REGION Network 13: Реле безопастности К21 группа 221,222,224,225,231-235,311,312,313-317
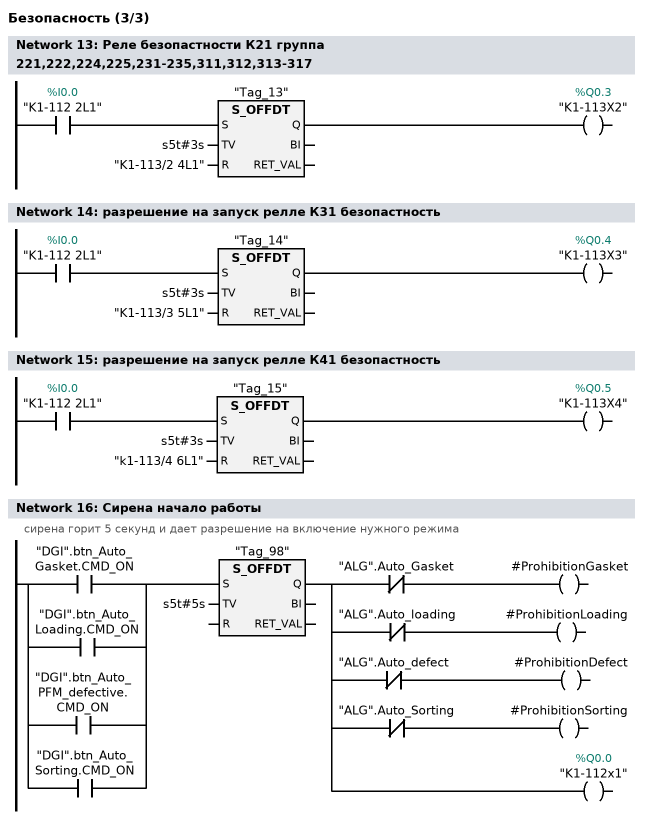
   RUNG wire#powerrail
      Contact( "K1-112 2L1" )
      S_OFFDT(T_NO := "Tag_13", TV := s5t#3s, R := "K1-113/2 4L1", BI =>, RET_VAL =>)
      Coil( "K1-113X2" )
   END_RUNG
   // the same network as SCL:
   #_s5time1 := S_OFFDT(T_NO := "Tag_13", S := "K1-112 2L1", TV := s5t#3s, R := "K1-113/2 4L1", Q => #_w1);
   "K1-113X2" := #_w1;
END_REGION

REGION Network 14: разрешение на запуск релле К31 безопастность
   RUNG wire#powerrail
      Contact( "K1-112 2L1" )
      S_OFFDT(T_NO := "Tag_14", TV := s5t#3s, R := "K1-113/3 5L1", BI =>, RET_VAL =>)
      Coil( "K1-113X3" )
   END_RUNG
   // the same network as SCL:
   #_s5time1 := S_OFFDT(T_NO := "Tag_14", S := "K1-112 2L1", TV := s5t#3s, R := "K1-113/3 5L1", Q => #_w1);
   "K1-113X3" := #_w1;
END_REGION

REGION Network 15: разрешение на запуск релле К41 безопастность
   RUNG wire#powerrail
      Contact( "K1-112 2L1" )
      S_OFFDT(T_NO := "Tag_15", TV := s5t#3s, R := "k1-113/4 6L1", BI =>, RET_VAL =>)
      Coil( "K1-113X4" )
   END_RUNG
   // the same network as SCL:
   #_s5time1 := S_OFFDT(T_NO := "Tag_15", S := "K1-112 2L1", TV := s5t#3s, R := "k1-113/4 6L1", Q => #_w1);
   "K1-113X4" := #_w1;
END_REGION

REGION Network 16: Сирена начало работы
   // сирена горит 5 секунд и дает разрешение на включение нужного режима
   RUNG wire#powerrail
      Contact( "DGI".btn_Auto_Gasket.CMD_ON )
      wire#w1
      S_OFFDT(T_NO := "Tag_98", TV := s5t#5s, R :=, BI =>, RET_VAL =>)
      wire#w2
      I_Contact( "ALG".Auto_Gasket )
      Coil( #ProhibitionGasket )
   END_RUNG
   RUNG wire#powerrail
      Contact( "DGI".btn_Auto_Loading.CMD_ON )
   END_RUNG wire#w1
   RUNG wire#powerrail
      Contact( "DGI".btn_Auto_PFM_defective.CMD_ON )
   END_RUNG wire#w1
   RUNG wire#powerrail
      Contact( "DGI".btn_Auto_Sorting.CMD_ON )
   END_RUNG wire#w1
   RUNG wire#w2
      I_Contact( "ALG".Auto_loading )
      Coil( #ProhibitionLoading )
   END_RUNG
   RUNG wire#w2
      I_Contact( "ALG".Auto_defect )
      Coil( #ProhibitionDefect )
   END_RUNG
   RUNG wire#w2
      I_Contact( "ALG".Auto_Sorting )
      Coil( #ProhibitionSorting )
   END_RUNG
   RUNG wire#w2
      Coil( "K1-112x1" )
   END_RUNG
   // the same network as SCL:
   #_s5time1 := S_OFFDT(T_NO := "Tag_98",
                        S := "DGI".btn_Auto_Gasket.CMD_ON OR "DGI".btn_Auto_Loading.CMD_ON OR "DGI".btn_Auto_PFM_defective.CMD_ON OR "DGI".btn_Auto_Sorting.CMD_ON,
                        TV := s5t#5s,
                        Q => #_w1);
   #ProhibitionGasket := #_w1 AND NOT "ALG".Auto_Gasket;
   #ProhibitionLoading := #_w1 AND NOT "ALG".Auto_loading;
   #ProhibitionDefect := #_w1 AND NOT "ALG".Auto_defect;
   #ProhibitionSorting := #_w1 AND NOT "ALG".Auto_Sorting;
   "K1-112x1" := #_w1;
END_REGION
END_FUNCTION_BLOCK

FUNCTION_BLOCK "FB_Link_Server"
{ S7_Optimized_Access := 'FALSE' }
VERSION : 0.1
   VAR 
      OperatorDetected : Bool;   // Можно начинать пересортировку оператор начал смену
      PackResortedReaded : Bool;   //     Пересортированный пакет прочитан
      FinishPackResorting : Bool;   //     Принудительно закончить пересортировку пакета
      Enable2Sxema : Bool;   // Собрать пакет 2мя схемами прокладок
      EnableRolling : Bool;   // Раскатать доски пакета на заданную длину
      SettingsWasApplyied : Bool;   // Были применены новые  настройки
      CheckPlankL : Bool;   // Проверять длину доски
      FinishDefectPack : Bool;   // Принудительно закончить сборку пакета  ПФМ брака
      DefectPacketPushed : Bool;   // пакет на ПФМ брака забрали
      PackDefectReaded : Bool;   // пакет на ПФМ брака прочитан сервером 
      PackParamChanged : Bool;   // Изменить параметры пакета
      PackReadyRidOff : Bool;   // пакет готов к выкатке
      GasketRidedOff : Bool;   // прокладку забрали с рамы
      PackToPack : Bool;   // режим из пакета в пакет
      AddGasketLayer : Bool;   // еще слой прокладки
      PackBrakParamChanged : Bool;   // корректировка параметров пакета брака
      QPlankLayers : Int;   // Количество слоев в пакете
      VPlanksInPack : Int;   //     Объём досок в пакете, м3
      QPlanksInLayer : Int;   //     Кол-во досок в слое досок пакета, шт
      QPlanksInLayerBrak : Int;   //     Кол-во досок в слое досок пакета брака, шт
      QPLankLayersBrak : Int;   //  Кол-во слоёв в пакете брака, шт
      Sxema : DInt;   //   Схема укладки прокладок
      SxemaNum : Int;   //     Номер схемы укладок прокладок
      PlankW : Int;   //     Ширина доски, мм
      PlankT : Int;   //     Толщина доски, мм
      Sxema2 : DInt;   // Cхема 2 укладки прокладок
      Sxema2Qlayers : Int;   //  Кол-во слоёв схемы 2 укладки прокладок
      PackL : Int;   // Длина пересобираемого пакета
      PartId : DInt;   // Ключ к пересобираемой партии (на случай перезапуска сервака)
      PlankL : Int;   // проверяемая длина доски
      ItemId : DInt;   // Ключ к номенклатуре пакета (на случай перезапуска сервака)
      SetNumLayer : Int;   // Корректируемое кол-во уложенных слоев досокб шт
      SetNumPlankInLayer : Int;   // Коррктируемое кол-во досок в слоеб шт
      GeneralSpeed : Int := 50;   // Общая скорость линии
      TotalPlanksInPack : Int;   // всего досок в пакете
      SetNumPlanksInLayerBrak : Int;   // коррекция счета досок в слое брака
      CheckL : Int;   // проверяемая длина доски
      GasketBrakPut : Bool;   // положили бруски на пакет брака
      GasketLayersPeriod : Int;   // Периодичность брусков пакета брака
      LineInWork : Bool;   //     Линия в работе
      PackResorting : Bool;   //     Пакет пересортировывается
      PackResorted : Bool;   //     Пакет пересортировался
      PackBrakComplete : Bool;   //  Пакет брака собран
      RdyStartNewPack : Bool;   //     Есть готовность к пересборке нового пакета
      RdyStart : Bool;   //     Есть готовность к запуску линии
      DefectPacketResorted : Bool;   // Пакет на ПФМ брака пересортирован
      NumLayerActual : Int;   //     Текущее кол-во уложенных слоёв досок, шт
      NumPlanksInLayerActual : Int;   //     Текущее кол-во уложенных слоёв прокладок, шт
      QPlanksOk : Int;   //     Текущее кол-во уложенных досок, шт
      QPlanksNotOk : Int;   //     Текущее кол-во уложенных херовых досок, шт
      VPlanksOk : DInt;   //     Текущий объём уложенных досок, м3*1000
      QPlankBrak : Int;   // Кол-во досок в пакете брака
      VLayerOk : DInt;   // Объем собирающегося слоя, м3
      M_211 : "ServIM";   //      Загрузочный транспортёр
      M_212 : "ServIM";   //      Загрузочный лифт сортировки+тормоз
      M_213 : "ServIM";   //      Наклюнный транспортёр после лифта
      M_214 : "ServIM";   //      Приёмный транспортёр прокладок
      M_221 : "ServIM";   //      Горка основная
      M_222 : "ServIM";   //      Транспортёр цепной после элеватора
      M_223 : "ServIM";   //      Резерв
      M_224 : "ServIM";   //      Упоры поштучника
      M_225 : "ServIM";   //      Транспортёр бобышек
      M_231 : "ServIM";   //      Ролики торцовочные
      M_232 : "ServIM";   //      Лифт ПФМ
      M_233 : "ServIM";   //      Вилы ПФМ
      ForkRotator : "ServIM";   //  Поворот вилы основной ПФМ
      M_234 : "ServIM";   //      Тр-тёр прокладок перед крючками ПФМ
      M_235 : "ServIM";   //      Подвижной борт
      M_311 : "ServIM";   //      Ленточный тр-тёр удаления прокладок
      M_312 : "ServIM";   //      Горка прокладок 1
      M_313 : "ServIM";   //      Тр-тёр прокладок после горки прокладок 1
      M_314 : "ServIM";   //      Горка прокладок 2
      M_315 : "ServIM";   //      Горка прокладок 3
      M_316 : "ServIM";   //      Тр-тёр загрузки прокладок в горку 2
      M_317 : "ServIM";   //      Основной транспортёр прокладок
      GasketSupplier : "ServIM";   // Выдача прокладки на карусель
      M_321 : "ServIM";   //      Выкатной транспортёр ПФМ 1
      M_322 : "ServIM";   //      Выкатной транспортёр ПФМ 2
      M_323 : "ServIM";
      M_324 : "ServIM";   //      Выкатной транспортёр ПФМ 3 (выгрузка пакета)
      M_325 : "ServIM";   //  Транспортер приема доски с Горки перед поштучкой
      M_330 : "ServIM";   //  Ленточный транспортер брака
      M_331 : "ServIM";   //      Ленточный транспортёр брака
      M_332 : "ServIM";   //      Сбрасыватель с рольганга брака
      M_333 : "ServIM";   //      Рольганг брака
      M_334 : "ServIM";   //      Тр-тёр сбора слоя ПФМ брака
      M_335 : "ServIM";   //      Вилы ПФМ брака
      M_336 : "ServIM";   //      Лифт ПФМ брака
      Alarm_List { S7_SetPoint := 'True'} : Array[0..255] of Bool;
   END_VAR


BEGIN
	    //Сбросим задание на подвижный борт, после того как в FB_Link_Server он был взведен по новому заданию
	    "ALG".ModeChang := FALSE;
	    "ALG".ForceFinishMainPFM := FALSE;
	    "ALG".ForceFinishPFMDefect := FALSE;
	    "ALG".DefectivePacketIsPushed := FALSE;
	    "ALG".EmptyLodems := FALSE;
	    "ALG".AddGasketLayer := FALSE;
	    "ALG".ConfirmGasketsBrak := FALSE;
	    
	    //Пришел бит с сервера "Начать новый пакет" (вместе с прочими исходными данными)
	 //   IF #OperatorDetected THEN
	 //       #QPlanksNotOk := 0;
	 //       #QPlanksOk := 0;
	        
	        // В конце бит с сервера "Начать новый пакет" обнулим
	 //       #OperatorDetected := FALSE;
	 //   END_IF;
	    
	    //Ежели были применены новые настройки
	    IF #SettingsWasApplyied THEN
	        
	      // для подвижного борта
	        "ALG".ModeChang := true;
	        
	        // для определения задержки
	        "ALG".PermMovM323 := "SolveLinearDelay"(LinearParam:=#PlankW, Koef:=2.5, Offset:=10);
	        "ALG".SqueezeRamp := "SolveLinearDelay"(LinearParam := 60 - #PlankT,
	                                                Koef := 10.0,
	                                                Offset := 100);
	        
	        "ALG".SqueezeUporPFM := "SolveLinearDelay"(LinearParam := #PlankT,
	                                                   Koef := 3.75,
	                                                   Offset := 10);
	        
	        #PackResorted := FALSE;
	        
	        #RdyStartNewPack := False;
	        
	        #RdyStart := FALSE;
	        #SettingsWasApplyied := FALSE;
	        
	       
	    END_IF;
	    
	    
	    
	    //Пришел бит с сервера или кнопки "Принудительно завершить пересортировку пакета"
	    IF #FinishPackResorting THEN
	        
	        //...//
	        "ALG".ForceFinishMainPFM := TRUE;
	        
	        // В конце его обнулим
	        #FinishPackResorting := FALSE;
	    END_IF;
	    
	    //Пришел бит с сервера "Принудительно завершить пересортировку пакета брака"
	    IF #FinishDefectPack THEN
	        
	        //...//
	        "ALG".ForceFinishPFMDefect := TRUE;
	        
	        
	        // В конце его обнулим
	        #FinishDefectPack := FALSE;
	    END_IF;
	    
	    IF (#DefectPacketPushed) THEN
	        "ALG".DefectivePacketIsPushed := TRUE;
	        
	        #DefectPacketPushed := FALSE;
	    END_IF;
	    
	    // Пришел битяра, что пакет брака прочитан и записан в ДБ
	    IF (#PackDefectReaded) THEN
	        
	        #DefectPacketResorted := FALSE;
	        #QPlanksNotOk := 0;
	        
	        #PackDefectReaded := False;
	    END_IF;
	    
	    // Пришел бит на изменение кол-ва досок в слое, кол-во слоев в пакете
	    IF (#PackParamChanged) THEN
	        // если на раме прокладок сейчас ничего нет, то просто меняем внутренний счетчик
	        IF ( "Сортировка_DB".LayersCounter <> #SetNumLayer) THEN
	            IF ("FB_Ramp_DB".s_busy) THEN
	                "FB_Ramp_DB".layer_holded := #SetNumLayer + 1;
	            ELSE
	                "FB_Ramp_DB".layer_holded := #SetNumLayer;
	            END_IF;
	        END_IF;
	        
	        "Сортировка_DB".LayersCounter := #SetNumLayer;
	        "Сортировка_DB".BoardInLayerCounter := #SetNumPlankInLayer;
	        
	        
	        
	        #PackParamChanged := False;
	    END_IF;
	    
	    
	    // На пакет наклеили этикетку
	    IF (#PackReadyRidOff) THEN
	        // Переменная для работы логики фиксируется
	        "ALG".PacketReadyRollOut := "S16.1" AND "B18.0" AND "Сортировка_DB".LiftPushingPacket;
	        // сразу обнуляемся
	        #PackReadyRidOff := FALSE;
	    END_IF;
	    
	    //бит прокладочник очищен
	    IF (#GasketRidedOff) THEN
	        "ALG".EmptyLodems := TRUE;
	        
	        #GasketRidedOff := FALSE;
	    END_IF;
	    
	    // бит добавить еще слой прокладок
	    // 
	    IF (#AddGasketLayer) THEN
	        "ALG".AddGasketLayer := TRUE;
	        
	        #AddGasketLayer := FALSE;
	    END_IF;
	    
	    IF (#GasketBrakPut) THEN
	        "ALG".ConfirmGasketsBrak := "B22.6";
	        
	        #GasketBrakPut := FALSE;
	    END_IF;
	   
	    //
	    IF (#PackBrakParamChanged) THEN
	        "ПФМ Брака_DB".BoardsInLayCounter := #SetNumPlanksInLayerBrak;
	        
	        #PackBrakParamChanged := FALSE;
	    END_IF;
	    
	    //Пришел бит с сервера "Сервер прочитал что пакет пересобран" или бит "Принудительно завершить пересортировку пакета"
	    IF #PackResortedReaded THEN
	        
	        //...// 
	        
	        //Обнулим задание на пересборку пакета и актуальные значения
	(*        #NumGasketActual := 0;
	        #NumLayerActual := 0;
	        #PlankT := 0;
	        #PlankW := 0;
	        #Sxema := 0;
	        #QPlanksInLayerBrak := 0;
	        #QPlankLayers := 0;
	        #QPlanksInLayer := 0;
	        #QPlanksNotOk := 0;
	        #QPlanksOk := 0;
	        #SxemaNum := 0;
	        #VPlanksOk := 0;
	        #Sxema2 := 0;
	        #Sxema2Qlayers := 0;
	        #PackL := 0; *)
	        //#PackId := 0;
	        //
	        #QPlanksOk := 0;
	        "ALG".Volume := 0;
	        #VPlanksOk := 0;
	        
	        #PackResorted := FALSE;
	        
	        // В конце его обнулим
	        #PackResortedReaded := FALSE;
	    END_IF;
	    //==============================================================================================
	    //M211 Загрузочный транспортер пакета
	    
	    (* IF #M_211.BtnAU THEN
	        #M_211.BtnAU := FALSE;
	    END_IF;
	    IF #M_211.BtnDU THEN
	        #M_211.BtnDU := FALSE;
	    END_IF;
	    IF #M_211.BtnFwd THEN
	        #M_211.BtnFwd := FALSE;
	    END_IF;
	    IF #M_211.BtnBwd THEN
	        #M_211.BtnBwd := FALSE;
	    END_IF;
	    IF #M_211.BtnCmdStop THEN
	        #M_211.BtnCmdStop := FALSE;
	    END_IF;     
	    IF #M_211.BtnDU THEN
	        "IM".M_211_Load_Transp.btnDU := TRUE;
	        #M_211.BtnDU := FALSE;
	        
	    END_IF;*)
	    
	    
	    REGION Список аварий заполнение
	        // Motor faults
	        // 
	        #Alarm_List[0] := "IM".M_211_Load_Transp.notON;
	        #Alarm_List[1] := "IM".M_211_Load_Transp.notOFF;
	        #Alarm_List[2] := "IM".M_311_Strip_Remov.notON;
	        #Alarm_List[3] := "IM".M_311_Strip_Remov.notOFF;
	        #Alarm_List[4] := "IM".M_212_Sort_Elevator.notOn;
	        #Alarm_List[5] := "IM".M_212_Sort_Elevator.notCMD;
	        #Alarm_List[6] := "IM".M_212_Sort_Elevator.notOff;
	        #Alarm_List[7] := "IM".M_212_Sort_Elevator.wrong_state;
	        #Alarm_List[8] := "IM".M_212_Sort_Elevator.wrong_CMD;
	        #Alarm_List[9] := "IM".M_213_ConvElevator.notON;
	        #Alarm_List[10] := "IM".M_213_ConvElevator.notOFF;
	        #Alarm_List[11] := "IM".M_222_Main_Sort_Slide.notON;
	        #Alarm_List[12] := "IM".M_222_Main_Sort_Slide.notOFF;
	        #Alarm_List[13] := "IM".M_325_Tr_Hill.notON;
	        #Alarm_List[14] := "IM".M_325_Tr_Hill.notOFF;
	        #Alarm_List[15] := "IM".M_223_Evaluation_area.notON;
	        #Alarm_List[16] := "IM".M_223_Evaluation_area.notOFF;
	        #Alarm_List[17] := "IM".M_224_Individ_dispensing.notOn;
	        #Alarm_List[18] := "IM".M_224_Individ_dispensing.notCMD;
	        #Alarm_List[19] := "IM".M_224_Individ_dispensing.notOff;
	        #Alarm_List[20] := "IM".M_224_Individ_dispensing.wrong_state;
	        #Alarm_List[21] := "IM".M_224_Individ_dispensing.wrong_CMD;
	        #Alarm_List[22] := "IM".M_225_Conveyor_with_lugs.notON;
	        #Alarm_List[23] := "IM".M_225_Conveyor_with_lugs.notOFF;
	        #Alarm_List[24] := "IM".M_235_Movable_board.notOn;
	        #Alarm_List[25] := "IM".M_235_Movable_board.notCMD;
	        #Alarm_List[26] := "IM".M_235_Movable_board.notOff;
	        #Alarm_List[27] := "IM".M_235_Movable_board.wrong_state;
	        #Alarm_List[28] := "IM".M_235_Movable_board.wrong_CMD;
	        #Alarm_List[29] := "IM".M_231_Roller_conveyor.notON;
	        #Alarm_List[30] := "IM".M_231_Roller_conveyor.notOFF;
	        #Alarm_List[31] := "IM".M_323_Small_Chain.notON;
	        #Alarm_List[32] := "IM".M_323_Small_Chain.notOFF;
	        #Alarm_List[33] := "IM".M_214_Gasket_receiver.notON;
	        #Alarm_List[34] := "IM".M_214_Gasket_receiver.notOFF;
	        #Alarm_List[35] := "IM".M_312_First_slide.notON;
	        #Alarm_List[36] := "IM".M_312_First_slide.notOFF;
	        #Alarm_List[37] := "IM".M_313_AF_slide_conv.notON;
	        #Alarm_List[38] := "IM".M_313_AF_slide_conv.notOFF;
	        #Alarm_List[39] := "IM".M_316_Padloader_IN2.notON;
	        #Alarm_List[40] := "IM".M_316_Padloader_IN2.notOFF;
	        #Alarm_List[41] := "IM".M_314_Second_slide.notON;
	        #Alarm_List[42] := "IM".M_314_Second_slide.notOFF;
	        #Alarm_List[43] := "IM".M_315_Third_slide.notON;
	        #Alarm_List[44] := "IM".M_315_Third_slide.notOFF;
	        #Alarm_List[45] := "IM".M_234_Carousel_loader.notON;
	        #Alarm_List[46] := "IM".M_234_Carousel_loader.notOFF;
	        #Alarm_List[47] := "IM".M_330_Scrap_Conv.notON;
	        #Alarm_List[48] := "IM".M_330_Scrap_Conv.notOFF;
	        #Alarm_List[49] := "IM".M_331_Scrap_conveyor.notON;
	        #Alarm_List[50] := "IM".M_331_Scrap_conveyor.notOFF;
	        #Alarm_List[51] := "IM".M_332_Dump_lug_conv.notON;
	        #Alarm_List[52] := "IM".M_332_Dump_lug_conv.notOFF;
	        #Alarm_List[53] := "IM".M_333_Defective_roller.notON;
	        #Alarm_List[54] := "IM".M_333_Defective_roller.notOFF;
	        #Alarm_List[55] := "IM".M_334_Layer_set_conv.notON;
	        #Alarm_List[56] := "IM".M_334_Layer_set_conv.notOFF;
	        #Alarm_List[57] := "IM".M_335_Lay_fork_scrap.notON;
	        #Alarm_List[58] := "IM".M_335_Lay_fork_scrap.notOFF;
	        #Alarm_List[59] := "IM".M_335_Lay_fork_scrap.notCMD;
	        #Alarm_List[60] := "IM".M_335_Lay_fork_scrap.notFeedBack;
	        #Alarm_List[61] := "IM".M_335_Lay_fork_scrap.wrong_state;
	        #Alarm_List[62] := "IM".M_336_PFM_elevator.notOn;
	        #Alarm_List[63] := "IM".M_336_PFM_elevator.notCMD;
	        #Alarm_List[64] := "IM".M_336_PFM_elevator.notOff;
	        #Alarm_List[65] := "IM".M_336_PFM_elevator.wrong_state;
	        #Alarm_List[66] := "IM".M_336_PFM_elevator.wrong_CMD;
	        #Alarm_List[67] := "IM_Rout".M_321_Rollgang_Lift_PFM.notON;
	        #Alarm_List[68] := "IM_Rout".M_321_Rollgang_Lift_PFM.notOFF;
	        #Alarm_List[69] := "IM_Rout".M_322_Conveyor_2.notON;
	        #Alarm_List[70] := "IM_Rout".M_322_Conveyor_2.notOFF;
	        #Alarm_List[71] := "IM_Rout".M_324_Rout_Conveyor.notON;
	        #Alarm_List[72] := "IM_Rout".M_324_Rout_Conveyor.notOFF;
	        #Alarm_List[73] := "IM_PFM".M_233_Fork_PFM.notON;
	        #Alarm_List[74] := "IM_PFM".M_233_Fork_PFM.notOFF;
	        #Alarm_List[75] := "IM_PFM".M_233_Fork_PFM.notCMD;
	        #Alarm_List[76] := "IM_PFM".M_233_Fork_PFM.notFeedBack;
	        #Alarm_List[77] := "IM_PFM".M_232_Elevator_PFM.notOn;
	        #Alarm_List[78] := "IM_PFM".M_232_Elevator_PFM.notCMD;
	        #Alarm_List[79] := "IM_PFM".M_232_Elevator_PFM.notOff;
	        #Alarm_List[80] := "IM_PFM".M_232_Elevator_PFM.wrong_state;
	        #Alarm_List[81] := "IM_PFM".M_232_Elevator_PFM.wrong_CMD;
	        #Alarm_List[82] := "IM_PFM".M_317_Gasket_Carousel.notON;
	        #Alarm_List[83] := "IM_PFM".M_317_Gasket_Carousel.notOFF;
	        #Alarm_List[84] := "HS".Gasket_Ramp.notUp;
	        #Alarm_List[85] := "HS".Gasket_Ramp.notMid;
	        #Alarm_List[86] := "HS".Gasket_Ramp.notDn;
	        #Alarm_List[87] := "HS".Gasket_Ramp.wrong_state;
	        #Alarm_List[88] := "HS".Gasket_Ramp.wrong_CMD;
	        #Alarm_List[89] := "HS".Gasket_Lodems.notON;
	        #Alarm_List[90] := "HS".Gasket_Lodems.notOFF;
	        #Alarm_List[91] := "HS".Gasket_Lodems.notCMD;
	        #Alarm_List[92] := "HS".Gasket_Lodems.notFeedBack;
	        #Alarm_List[93] := "HS".Gasket_Lodems.wrong_state;
	        #Alarm_List[94] := "HS".Forks_Pitcher.notON;
	        #Alarm_List[95] := "HS".Forks_Pitcher.notOFF;
	        #Alarm_List[96] := "HS".Forks_Pitcher.notCMD;
	        #Alarm_List[97] := "HS".Forks_Pitcher.notFeedBack;
	        #Alarm_List[98] := "HS".Forks_Pitcher.wrong_state;
	        #Alarm_List[99] := "HS".Upor_Defective.notON;
	        #Alarm_List[100] := "HS".Upor_Defective.notOFF;
	        #Alarm_List[101] := "HS".Upor_Defective.notCMD;
	        #Alarm_List[102] := "HS".Upor_Defective.notFeedBack;
	        #Alarm_List[103] := "HS".Upor_Defective.wrong_state;
	        #Alarm_List[104] := "HS".M_221_Large_HydroStationDrive.notOn;
	        #Alarm_List[105] := "HS".M_221_Large_HydroStationDrive.notOff;
	        #Alarm_List[106] := "HS".M_221_Large_HydroStationDrive.wrongValveState;
	        #Alarm_List[107] := "HS".M_337_Small_HydroStationDrive.notOn;
	        #Alarm_List[108] := "HS".M_337_Small_HydroStationDrive.notOff;
	        #Alarm_List[109] := "HS".M_337_Small_HydroStationDrive.wrongValveState;
	        
	        
	        // Logic faults
	        // 
	        #Alarm_List[110] := "QueueController_DB".AlarmWrongLength;
	        #Alarm_List[111] := "FB_Gasket_Carousel_DB".s_paused; // "FB_SetGaskets_DB".Paused;
	        #Alarm_List[112] := "FB_Gasket_Carousel_DB".ALM_NoGasketToUP;  // "FB_SetGaskets_DB".ALM_NoGasketToUP;
	        #Alarm_List[113] := "EvaluationZoneThrowOFF_DB".AlarmBoardNotExitFromZone;
	        #Alarm_List[114] := "Сортировка_DB".AlarmLowerElevator;
	        #Alarm_List[115] := "UporPFM_DB".AlarmGidra; // уберите доску после упоров ПФМ
	        #Alarm_List[116] := "UporPFM_DB".AlarmWarpingBoard; // уберите доску после упоров ПФМ
	        
	        // Sxema Faults
	        // 
	        
	        #Alarm_List[117] := "QueueController_DB".AlarmNotValidHole AND NOT "QueueController_DB".Hint_3;  // Ожидался пробел между слоями, уберите доску под линейкой, следующая доска должна быть на низкой цепи
	        #Alarm_List[118] := "QueueController_DB".AlarmNotValidHole AND "QueueController_DB".Hint_3;
	        
	        #Alarm_List[119] := "QueueController_DB".AlarmNotAwaitableBoard AND "QueueController_DB".Hint_3 AND NOT "QueueController_DB".Hint_2; // не та доска под линейкой, переложите на след бобышку, следующая цепь высокая (Далее ожидается доска на высокой цепи)
	        #Alarm_List[120] := "QueueController_DB".AlarmNotAwaitableBoard AND "QueueController_DB".Hint_3  AND "QueueController_DB".Hint_2; // под линейкой ожидалась доска на высокой цепи, уберите доску
	        #Alarm_List[121] := "QueueController_DB".AlarmNotAwaitableBoard AND NOT "QueueController_DB".Hint_3  AND "QueueController_DB".Hint_2; // под линейкой ожидалась доска на низкой цепи, уберите доску
	        
	        #Alarm_List[122] := "QueueController_DB".AlarmNotAwaitableBoard AND NOT "QueueController_DB".Hint_3 AND NOT "QueueController_DB".Hint_2; // не та доска под линейкой, переложите на след бобышку, следующая цепь низкая Далее ожидается доска на низкой цепи)
	        
	        // SensLineAlarm
	        // 
	        #Alarm_List[123] := "SensorLine_Clogging_DB".AlarmSensor_dirty[0]; //загрязнен датчик 1,8 м
	        #Alarm_List[124] := "SensorLine_Clogging_DB".AlarmSensor_dirty[1];
	        #Alarm_List[125] := "SensorLine_Clogging_DB".AlarmSensor_dirty[2];
	        #Alarm_List[126] := "SensorLine_Clogging_DB".AlarmSensor_dirty[3];
	        #Alarm_List[127] := "SensorLine_Clogging_DB".AlarmSensor_dirty[4];
	        #Alarm_List[128] := "SensorLine_Clogging_DB".AlarmSensor_dirty[5];
	        #Alarm_List[129] := "SensorLine_Clogging_DB".AlarmSensor_dirty[6];
	        #Alarm_List[130] := "SensorLine_Clogging_DB".AlarmSensor_dirty[7];
	        #Alarm_List[131] := "SensorLine_Clogging_DB".AlarmSensor_dirty[8];
	        #Alarm_List[132] := "SensorLine_Clogging_DB".AlarmSensor_dirty[9];
	        #Alarm_List[133] := "SensorLine_Clogging_DB".AlarmSensor_dirty[10];
	        #Alarm_List[134] := "SensorLine_Clogging_DB".AlarmSensor_dirty[11];
	        #Alarm_List[135] := "SensorLine_Clogging_DB".AlarmSensor_dirty[12];
	        #Alarm_List[136] := "SensorLine_Clogging_DB".AlarmSensor_dirty[13];
	        #Alarm_List[137] := "SensorLine_Clogging_DB".AlarmSensor_dirty[14]; // загрязнен датчик 6.0 м
	        
	        //Sensor alarms
	        //
	        
	        
	        //MOOOre alarms
	        // 
	        #Alarm_List[138] := "IM_PFM".M_233_Fork_PFM.unkn_state; // вилы ПФМ в некорректном положении
	        #Alarm_List[139] := "EvaluationZoneThrowOFF_DB".FaultGhostBoard; // ошибка очереди на зоне оценки
	        #Alarm_List[140] := NOT "QueueController_DB".Calibrated; // линейка не откалибрована
	        #Alarm_List[141] := "Сортировка_DB".AlarmNotReadedPack; // ошибка чтения пакета ПФМ
	        #Alarm_List[142] := "ПФМ Брака_DB".AlarmNotReadedPack; // ошибка чтения пакета ПФМ брака
	        #Alarm_List[143] := "ПФМ Брака_DB".AlarmExtraBoardInLay; //ошибка лишняя доска на слой пфм брака
	        #Alarm_List[144] := "FB_Gasket_Carousel_DB".ALM_SensLastHook;  // "FB_SetGaskets_DB".ALM_LargeOffset; // ошибка переезда карусели
	        #Alarm_List[145] := "FB_Gasket_Carousel_DB".ALM_SensHook; // "FB_SetGaskets_DB".ALM_SensHook; // сбой датчика крюков на карусели
	        #Alarm_List[146] := "QueueController_DB".AlarmCount; // ошибка счета ПФМ
	        #Alarm_List[147] := "ПФМ Брака_DB".AlarmNoPacketPushed; //авария не забрали пакет с пфм брака
	        #Alarm_List[148] := "ПФМ Брака_DB".AwaitGasket; // ожидаем прокладку на пфм брака
	        
	        
	    END_REGION
	    
	
END_FUNCTION_BLOCK

FUNCTION "SolveLinearDelay" : Time
{ S7_Optimized_Access := 'FALSE' }
VERSION : 0.1
   VAR_INPUT 
      LinearParam : Int;   // линейный параметр
      Koef : Real;   // коэффициент k
      Offset : Int;   // коэффициент сдвига b
   END_VAR

   VAR_TEMP 
      Delay_in_ms : Real;
   END_VAR


BEGIN
	#Delay_in_ms := INT_TO_REAL(#LinearParam);
	
	#SolveLinearDelay := DINT_TO_TIME(TRUNC_DINT(#Koef * #Delay_in_ms) + #Offset);
END_FUNCTION

FUNCTION "GetGeneralSpeed" : Real
{ S7_Optimized_Access := 'FALSE' }
VERSION : 0.1
   VAR_INPUT 
      GS_from_Server : Int;
   END_VAR


BEGIN
	IF (#GS_from_Server < 10.0) THEN
	    #GetGeneralSpeed := 10.0;
	ELSE
	    #GetGeneralSpeed := INT_TO_REAL(#GS_from_Server);
	END_IF;
	
END_FUNCTION

FUNCTION_BLOCK "FB_Load_Zone"
{ S7_Optimized_Access := 'FALSE' }
VERSION : 0.1
   VAR 
      auto_mode_trigger : Bool;
      M213_mode : Bool;
      up_cmd_old : Bool;
      down_cmd_old : Bool;
      Lift_State : Int;
      Memento_Lift_State : Int;
      delayStart {InstructionName := 'TON'; LibVersion := '1.0'} : TON;
      wait_1 {InstructionName := 'TOF'; LibVersion := '1.0'} : TOF;
      wait_2 {InstructionName := 'TOF'; LibVersion := '1.0'} : TOF;
      wait_3 {InstructionName := 'TOF'; LibVersion := '1.0'} : TOF;
      wait_213 {InstructionName := 'TOF'; LibVersion := '1.0'} : TOF;
   END_VAR

   VAR_TEMP 
      Lift_UP : Bool;
      Lift_DOWN : Bool;
      Cancel_UP : Bool;
      Resume_UP : Bool;
      Sert : Word;
   END_VAR

   VAR CONSTANT 
      LIFT_WAITING : Int := 0;
      LIFT_START : Int := 1;
      LIFT_CYCLE : Int := 2;
      LIFT_RETURN : Int := 3;
      LIFT_STOP : Int := 4;
      LIFT_CANCEL : Int := 5;
      LIFT_UNKNOWN : Int := 10;
      DELAY_START : Time := T#5s;
   END_VAR


BEGIN
	REGION Ready and alarms LOADING ZONE
	    
	    "ALG".Ready_loading := "NaprUpr" AND "K1-113/1 3L1" AND "K1-112 2L1";
	  
	    "ALG".Alarm_loading :=
	    // Транспортер загрузки
	    "IM".M_211_Load_Transp.Alarm OR
	    "IM".M_211_Load_Transp.Fault OR
	    // Лифт Melektra
	    "IM".M_212_Sort_Elevator.Fault OR
	    // Наклонный транспортер
	    "IM".M_213_ConvElevator.Fault OR
	    "IM".M_213_ConvElevator.Alarm OR
	    // Транспортер прокладок
	    "IM".M_214_Gasket_receiver.Fault OR
	    "IM".M_214_Gasket_receiver.Alarm OR
	    // ??
	    "IM".M_311_Strip_Remov.Fault OR
	    // НЕТ СИГНАЛА ГОТОВОСТИ
	    NOT "ALG".Ready_loading
	    ;
	    
	END_REGION
	
	REGION Mode selector
	    
	    #auto_mode_trigger := (#auto_mode_trigger
	    OR
	    (
	    "DGI".btn_Auto_Loading.CMD_ON
	    ))
	    AND NOT
	    (
	    NOT "ALG".Ready_loading OR
	    "DGI".btn_Auto_Loading.CMD_OFF
	    );
	    
	    // State lamps
	    // 
	    "H76.3" := "H78.0" := #auto_mode_trigger;
	    
	    // Auto SIGNAL
	    "ALG".Auto_loading := #auto_mode_trigger AND NOT "Безопасность_DB".ProhibitionLoading;
	    
	END_REGION
	
	REGION M211
	    // Backwards
	    "IM".M_211_Load_Transp.btn_Back_ON := "E82.2";
	    
	    // Forward
	    "IM".M_211_Load_Transp.OnCom :=
	    
	    "S81.1"
	    OR
	    ("IM".M_211_Load_Transp.btn_Back_ON)
	    ;
	    
	    
	END_REGION
	
	REGION M212
	    // SIGNALS
	    // 
	    #Cancel_UP := "DGI".E82_5 AND NOT #down_cmd_old;
	    #Resume_UP := "DGI".S82_4 AND NOT #up_cmd_old;
	    
	    #up_cmd_old := "DGI".S82_4;
	    #down_cmd_old := "DGI".E82_5;
	    
	    // таймера
	    // 
	    #delayStart(IN := "koncevik2",
	                PT := #DELAY_START);
	    
	    #wait_1(IN := "nakloniy transporter",
	            PT := T#6s);
	    
	    #wait_2(IN := NOT "doska v priymke elevator",
	            PT := T#3s);
	    
	    #wait_3(IN := "sloi doski",
	            PT := T#6s);
	    
	    
	    // запуск лифта
	    CASE #Lift_State OF
	        // ожидание пакета
	        #LIFT_WAITING:
	            
	            // LOGIC
	            #Lift_UP := #Lift_DOWN := FALSE;
	            //"IM".M_212_Sort_Elevator.comUp := "IM".M_212_Sort_Elevator.comDown := FALSE;
	            
	            // Transitions
	            IF (#delayStart.Q) THEN
	                #Lift_State := #LIFT_START;
	                GOTO EndAutomata;
	            END_IF;
	            
	            IF (NOT "Lift Down") THEN
	                #Lift_State := #LIFT_CANCEL;
	            END_IF;
	            
	        #LIFT_START:
	            
	            // LOGIC
	            // 
	            #Lift_UP := TRUE;
	            #Lift_DOWN := FALSE;
	            //"IM".M_212_Sort_Elevator.comUp := #delayStart.Q;
	            //"IM".M_212_Sort_Elevator.comDown := False;
	            
	            // Transitions
	            IF ("sloi doski") THEN
	                #Lift_State := #LIFT_CYCLE;
	                GOTO EndAutomata;
	            END_IF;
	            
	            IF ("Lift Upp") THEN
	                #Lift_State := #LIFT_RETURN;
	            END_IF;
	            
	            IF (#Cancel_UP) THEN
	                #Memento_Lift_State := #Lift_State;
	                #Lift_State := #LIFT_STOP;
	            END_IF;
	            
	        #LIFT_CYCLE:
	            // LOGIC
	            // 
	            #Lift_DOWN := FALSE;
	            #Lift_UP := NOT (#wait_1.Q OR #wait_2.Q OR #wait_3.Q) OR "DGI".S82_4;
	            
	            // Transitions
	            IF ("Lift Upp") THEN
	                #Lift_State := #LIFT_RETURN;
	            END_IF;
	            
	            IF (#Cancel_UP) THEN
	                #Memento_Lift_State := #Lift_State;
	                #Lift_State := #LIFT_STOP;
	            END_IF;
	            
	        #LIFT_RETURN:
	            // LOGIC
	            #Lift_DOWN := TRUE;
	            #Lift_UP := FALSE;
	            
	            // Transitions
	            IF ("Lift Down") THEN
	                #Lift_State := #LIFT_WAITING;
	                GOTO EndAutomata;
	            END_IF;
	            
	        #LIFT_STOP:
	            // LOGIC;
	            // 
	            #Lift_DOWN := FALSE;
	            #Lift_UP := False;
	            
	            // Transitions
	            // 
	            IF (#Cancel_UP) THEN
	                #Lift_State := #LIFT_CANCEL;
	                GOTO EndAutomata;
	            END_IF;
	            
	            IF (#Resume_UP) THEN
	               
	                #Lift_State := #Memento_Lift_State;
	                
	            END_IF;
	            
	        #LIFT_CANCEL:
	            // LOGIC
	            #Lift_DOWN := TRUE;
	            #Lift_UP := FALSE;
	            
	            // Transitions
	            IF ("Lift Down") THEN
	                #Lift_State := #LIFT_WAITING;
	                GOTO EndAutomata;
	            END_IF;
	
	        ELSE  // Lift unknown state
	            ;
	    END_CASE;
	    
	EndAutomata:
	    "IM".M_212_Sort_Elevator.comDown := NOT "ALG".Alarm_loading AND #Lift_DOWN;
	    "IM".M_212_Sort_Elevator.comUp := NOT "ALG".Alarm_loading AND #Lift_UP;
	    
	    IF ("IM".M_212_Sort_Elevator.outFWD) THEN
	        "IM".M_212_Sort_Elevator.setSpeedAU := "SolveSpeed"(GeneralSpeed:="VELOCITY".GeneralSpeed, MotorKoef:="VELOCITY".koef_M_212, Correction:=0.0);
	    ELSIF ("IM".M_212_Sort_Elevator.outBKD) THEN
	        IF (#Lift_State = #LIFT_RETURN) THEN
	            "IM".M_212_Sort_Elevator.setSpeedAU := 44.0;
	        ELSE
	            "IM".M_212_Sort_Elevator.setSpeedAU := 27.0;
	            
	        END_IF;
	    ELSE
	        "IM".M_212_Sort_Elevator.setSpeedAU := 0.0;
	    END_IF;
	    
	    #Sert := UNSCALE(IN := "IM".M_212_Sort_Elevator.setSpeed, HI_LIM := 50.0, LO_LIM := -50.0, BIPOLAR := TRUE, OUT => "K1-212U":P);
	    
	    
	END_REGION
	
	
	REGION M213
	    
	    REGION Selector Mode 
	        #M213_mode := "ServDB".PlankT <= 30;
	        
	        #wait_213(IN:=NOT "doska v priymke elevator",
	                  PT:=T#5s);
	        
	    END_REGION
	    
	    "IM".M_213_ConvElevator.OnCom := NOT "ALG".Alarm_loading AND
	    (
	    (#M213_mode AND NOT #wait_213.Q)
	    OR
	    (NOT #M213_mode AND "doska v priymke elevator")
	    );
	    
	    IF ("IM".M_213_ConvElevator.onOutFWD) THEN
	        "IM".M_213_ConvElevator.setSpeedAU := "SolveSpeed"(GeneralSpeed := "VELOCITY".GeneralSpeed, MotorKoef := "VELOCITY".koef_M_213, Correction := 0.0);
	    ELSE
	        "IM".M_213_ConvElevator.setSpeedAU := 0.0;
	    END_IF;
	    
	    #Sert := UNSCALE(IN := "IM".M_213_ConvElevator.setSpeed, HI_LIM := 50.0, LO_LIM := 0.0, BIPOLAR := FALSE, OUT => "K1-213U":P);
	        
	    
	END_REGION
	
END_FUNCTION_BLOCK

FUNCTION "SolveSpeed" : Real
{ S7_Optimized_Access := 'FALSE' }
VERSION : 0.1
   VAR_INPUT 
      GeneralSpeed : Real;   // общая скорость линии
      MotorKoef : Real;   // Коэффициент мотора
      Correction : Real;
   END_VAR


BEGIN
	#SolveSpeed := #GeneralSpeed * #MotorKoef + #Correction;
END_FUNCTION

FUNCTION_BLOCK "ПФМ Брака"   // FB3, LAD
VERSION : 0.1
// логика работы ПФМ брака
// stored: AutoNumber true, IsIECCheckEnabled false, UDAEnableTagReadback false
   VAR DB_SPECIFIC
      Trig332 : Bool;   // Тригер М332 сброс доски
      "TrigS79.3" : Bool;   // Тригер Авто режима
      ForcingPacket : Bool;
      LiftPushingPacket : Bool;   // лифт занят
      HodVil2 { ExternalAccessible := 'False'; ExternalVisible := 'False'; ExternalWritable := 'False'} : Bool;   // Триггер ход вил М335
      HodVil { ExternalAccessible := 'False'; ExternalVisible := 'False'; ExternalWritable := 'False'} : Bool;   // Триггер ход вил М335
      ForcingLift : Bool;
      CountSensor_front : Bool;
      StopDovod : Bool;
      StopDropppingBoards : Bool;
      newBob_old : Bool;
      liftDown_old : Bool;
      liftPushingPacket_old : Bool;
      newBoard_old : Bool;
      Upor_Off_trig : Bool;
      Lift_GoToStartPosition : Bool;
      ReviveSignal : Bool;   // сигнал для оживления механизмов
      StartAwaitForGasket : Bool;   // ожидание прокладок
      AwaitGasket : Bool;
      AlarmNotReadedPack : Bool;
      AlarmExtraBoardInLay : Bool;   // авария лишняя доска на слой ПФМ брака
      AlarmNoPacketPushed : Bool;
      BoardsInLayCounter : Int;   // Сравнение счетчика 2
      LayersCounter : Int;   // Счет слоев досок
   END_VAR
   VAR
      Board_counter : "Adder";   // Счетчик досок в слое
      Lay_counter : "Adder";   // Счетчик слоев
   END_VAR
   VAR_TEMP
      start_await : Bool;
      Sert : Word;
   END_VAR
   VAR_TEMP   // added for the SCL form of the ladder/FBD networks
      _w1 : Bool;
      _w2 : Bool;
      _w3 : Bool;
      _s5time1 : S5Time;
   END_VAR
BEGIN

REGION Network 1: Реле безопасности К41 группа 331,332-337
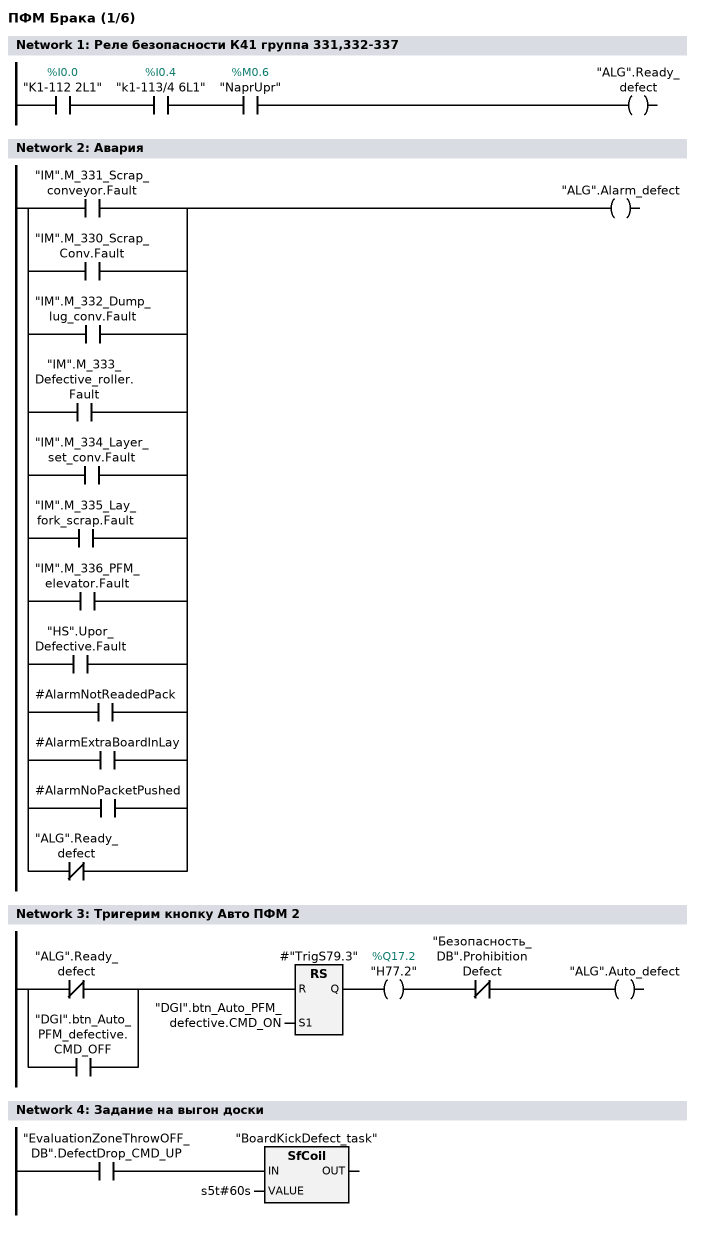
   RUNG wire#powerrail
      Contact( "K1-112 2L1" )
      Contact( "k1-113/4 6L1" )
      Contact( "NaprUpr" )
      Coil( "ALG".Ready_defect )
   END_RUNG
   // the same network as SCL:
   "ALG".Ready_defect := "K1-112 2L1" AND "k1-113/4 6L1" AND "NaprUpr";
END_REGION

REGION Network 2: Авария
   RUNG wire#powerrail
      Contact( "IM".M_331_Scrap_conveyor.Fault )
      wire#w1
      Coil( "ALG".Alarm_defect )
   END_RUNG
   RUNG wire#powerrail
      Contact( "IM".M_330_Scrap_Conv.Fault )
   END_RUNG wire#w1
   RUNG wire#powerrail
      Contact( "IM".M_332_Dump_lug_conv.Fault )
   END_RUNG wire#w1
   RUNG wire#powerrail
      Contact( "IM".M_333_Defective_roller.Fault )
   END_RUNG wire#w1
   RUNG wire#powerrail
      Contact( "IM".M_334_Layer_set_conv.Fault )
   END_RUNG wire#w1
   RUNG wire#powerrail
      Contact( "IM".M_335_Lay_fork_scrap.Fault )
   END_RUNG wire#w1
   RUNG wire#powerrail
      Contact( "IM".M_336_PFM_elevator.Fault )
   END_RUNG wire#w1
   RUNG wire#powerrail
      Contact( "HS".Upor_Defective.Fault )
   END_RUNG wire#w1
   RUNG wire#powerrail
      Contact( #AlarmNotReadedPack )
   END_RUNG wire#w1
   RUNG wire#powerrail
      Contact( #AlarmExtraBoardInLay )
   END_RUNG wire#w1
   RUNG wire#powerrail
      Contact( #AlarmNoPacketPushed )
   END_RUNG wire#w1
   RUNG wire#powerrail
      I_Contact( "ALG".Ready_defect )
   END_RUNG wire#w1
   // the same network as SCL:
   "ALG".Alarm_defect := "IM".M_331_Scrap_conveyor.Fault OR "IM".M_330_Scrap_Conv.Fault OR "IM".M_332_Dump_lug_conv.Fault OR "IM".M_333_Defective_roller.Fault OR "IM".M_334_Layer_set_conv.Fault OR "IM".M_335_Lay_fork_scrap.Fault OR "IM".M_336_PFM_elevator.Fault OR "HS".Upor_Defective.Fault OR #AlarmNotReadedPack OR #AlarmExtraBoardInLay OR #AlarmNoPacketPushed OR NOT "ALG".Ready_defect;
END_REGION

REGION Network 3: Тригерим кнопку Авто ПФМ 2
   RUNG wire#powerrail
      I_Contact( "ALG".Ready_defect )
      wire#w1
      S_RS(operand := #"TrigS79.3", s1 := "DGI".btn_Auto_PFM_defective.CMD_ON)
      Coil( "H77.2" )
      I_Contact( "Безопасность_DB".ProhibitionDefect )
      Coil( "ALG".Auto_defect )
   END_RUNG
   RUNG wire#powerrail
      Contact( "DGI".btn_Auto_PFM_defective.CMD_OFF )
   END_RUNG wire#w1
   // the same network as SCL:
   IF NOT "ALG".Ready_defect OR "DGI".btn_Auto_PFM_defective.CMD_OFF THEN
       #"TrigS79.3" := FALSE;   // RS flip-flop
   END_IF;
   IF "DGI".btn_Auto_PFM_defective.CMD_ON THEN #"TrigS79.3" := TRUE; END_IF;
   "H77.2" := #"TrigS79.3";
   "ALG".Auto_defect := #"TrigS79.3" AND NOT "Безопасность_DB".ProhibitionDefect;
END_REGION

REGION Network 4: Задание на выгон доски
   // no SCL statement known for SfCoil: written as a call
   SfCoil(in := "EvaluationZoneThrowOFF_DB".DefectDrop_CMD_UP,
          value := s5t#60s,
          operand := "BoardKickDefect_task");
END_REGION

REGION Network 5: Авто вперед М331/ M330
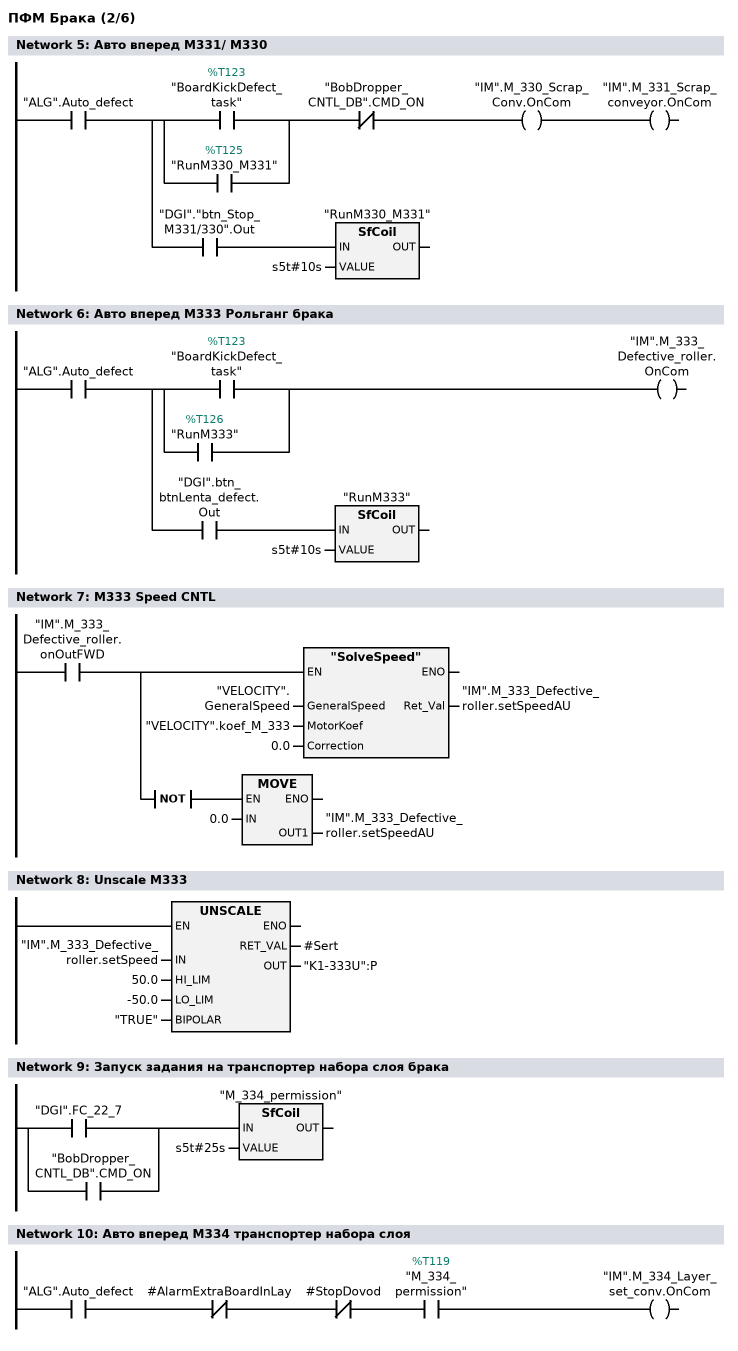
   // no SCL statement known for SfCoil: written as a call
   "IM".M_330_Scrap_Conv.OnCom := "ALG".Auto_defect AND ("BoardKickDefect_task" OR "RunM330_M331") AND NOT "BobDropper_CNTL_DB".CMD_ON;
   "IM".M_331_Scrap_conveyor.OnCom := "IM".M_330_Scrap_Conv.OnCom;
   SfCoil(in := "ALG".Auto_defect AND "DGI"."btn_Stop_M331/330".Out,
          value := s5t#10s,
          operand := "RunM330_M331");
END_REGION

REGION Network 6: Авто вперед М333 Рольганг брака
   // no SCL statement known for SfCoil: written as a call
   "IM".M_333_Defective_roller.OnCom := "ALG".Auto_defect AND ("BoardKickDefect_task" OR "RunM333");
   SfCoil(in := "ALG".Auto_defect AND "DGI".btn_btnLenta_defect.Out, value := s5t#10s, operand := "RunM333");
END_REGION

REGION Network 7: М333 Speed CNTL
   RUNG wire#powerrail
      Contact( "IM".M_333_Defective_roller.onOutFWD )
      wire#w1
      "SolveSpeed"(GeneralSpeed := "VELOCITY".GeneralSpeed, MotorKoef := "VELOCITY".koef_M_333, Correction := 0.0, Ret_Val => "IM".M_333_Defective_roller.setSpeedAU)
   END_RUNG
   RUNG wire#w1
      Not()
      { S7_GenerateENO := "TRUE" } Move(in := 0.0, out1 => "IM".M_333_Defective_roller.setSpeedAU)
   END_RUNG
   // the same network as SCL:
   #_w1 := "IM".M_333_Defective_roller.onOutFWD;
   IF #_w1 THEN
       "IM".M_333_Defective_roller.setSpeedAU := "SolveSpeed"(GeneralSpeed := "VELOCITY".GeneralSpeed,
                               MotorKoef := "VELOCITY".koef_M_333,
                               Correction := 0.0);
   END_IF;
   IF NOT #_w1 THEN "IM".M_333_Defective_roller.setSpeedAU := 0.0; END_IF;
END_REGION

REGION Network 8: Unscale M333
   RUNG wire#powerrail
      UNSCALE(IN := "IM".M_333_Defective_roller.setSpeed, HI_LIM := 50.0, LO_LIM := -50.0, BIPOLAR := "TRUE", RET_VAL => #Sert, OUT => "K1-333U":P)
   END_RUNG
   // the same network as SCL:
   #Sert := UNSCALE(IN := "IM".M_333_Defective_roller.setSpeed,
                    HI_LIM := 50.0,
                    LO_LIM := -50.0,
                    BIPOLAR := "TRUE",
                    OUT => "K1-333U":P);
END_REGION

REGION Network 9: Запуск задания на транспортер набора слоя брака
   // no SCL statement known for SfCoil: written as a call
   SfCoil(in := "DGI".FC_22_7 OR "BobDropper_CNTL_DB".CMD_ON, value := s5t#25s, operand := "M_334_permission");
END_REGION

REGION Network 10: Авто вперед М334 транспортер набора слоя
   RUNG wire#powerrail
      Contact( "ALG".Auto_defect )
      I_Contact( #AlarmExtraBoardInLay )
      I_Contact( #StopDovod )
      Contact( "M_334_permission" )
      Coil( "IM".M_334_Layer_set_conv.OnCom )
   END_RUNG
   // the same network as SCL:
   "IM".M_334_Layer_set_conv.OnCom := "ALG".Auto_defect AND NOT #AlarmExtraBoardInLay AND NOT #StopDovod AND "M_334_permission";
END_REGION

REGION Network 11: М334 транспортер набора слоя команды на движение
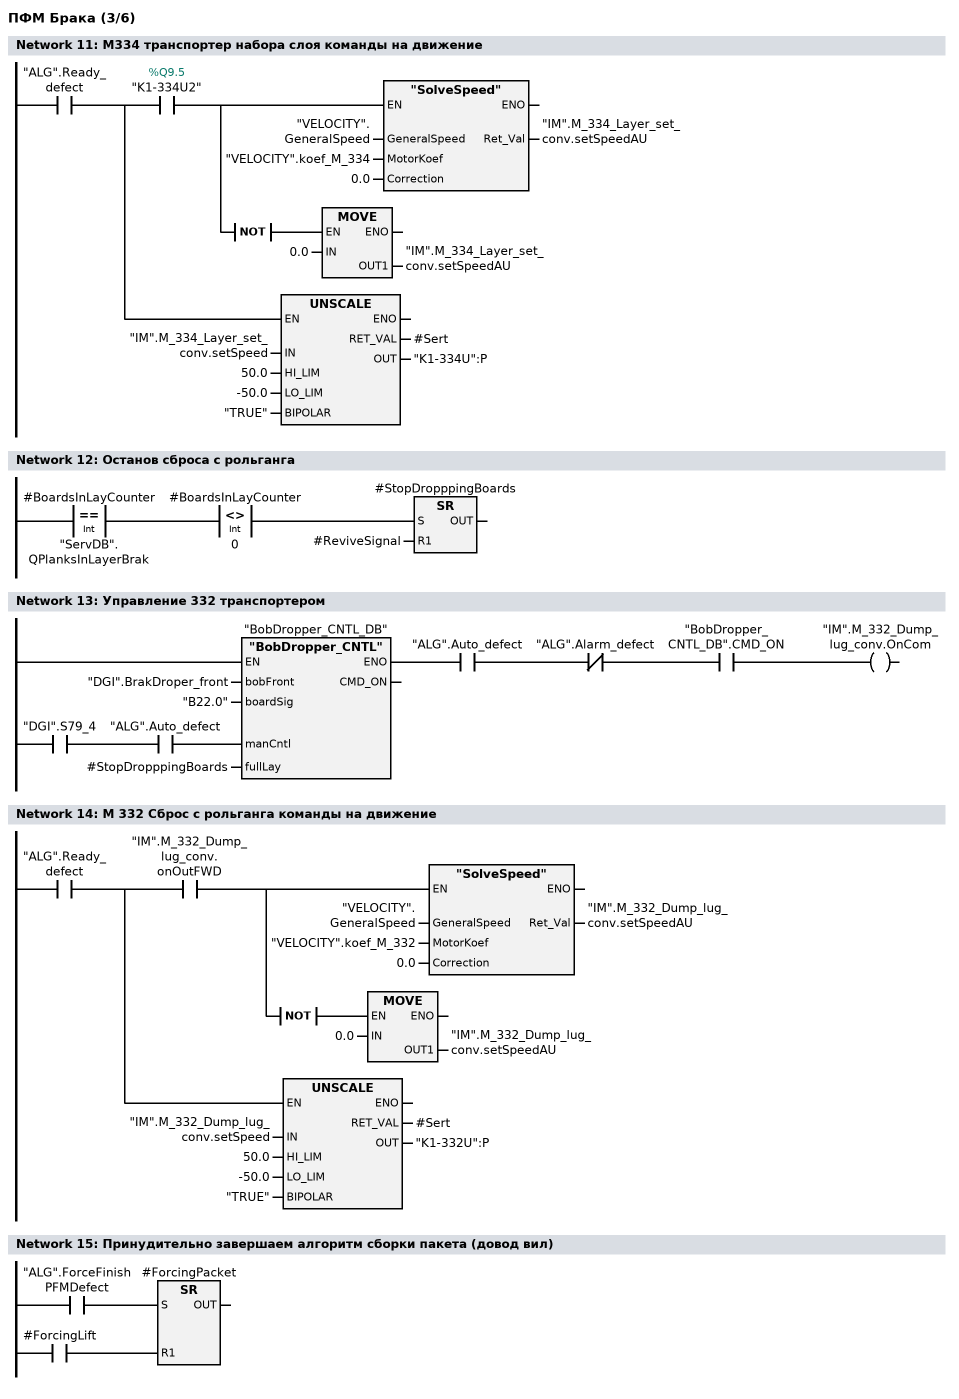
   RUNG wire#powerrail
      Contact( "ALG".Ready_defect )
      wire#w1
      Contact( "K1-334U2" )
      wire#w2
      "SolveSpeed"(GeneralSpeed := "VELOCITY".GeneralSpeed, MotorKoef := "VELOCITY".koef_M_334, Correction := 0.0, Ret_Val => "IM".M_334_Layer_set_conv.setSpeedAU)
   END_RUNG
   RUNG wire#w2
      Not()
      { S7_GenerateENO := "TRUE" } Move(in := 0.0, out1 => "IM".M_334_Layer_set_conv.setSpeedAU)
   END_RUNG
   RUNG wire#w1
      UNSCALE(IN := "IM".M_334_Layer_set_conv.setSpeed, HI_LIM := 50.0, LO_LIM := -50.0, BIPOLAR := "TRUE", RET_VAL => #Sert, OUT => "K1-334U":P)
   END_RUNG
   // the same network as SCL:
   #_w1 := "ALG".Ready_defect AND "K1-334U2";
   #_w2 := "ALG".Ready_defect;
   IF #_w1 THEN
       "IM".M_334_Layer_set_conv.setSpeedAU := "SolveSpeed"(GeneralSpeed := "VELOCITY".GeneralSpeed,
                               MotorKoef := "VELOCITY".koef_M_334,
                               Correction := 0.0);
   END_IF;
   IF NOT #_w1 THEN "IM".M_334_Layer_set_conv.setSpeedAU := 0.0; END_IF;
   IF #_w2 THEN
       #Sert := UNSCALE(IN := "IM".M_334_Layer_set_conv.setSpeed,
                        HI_LIM := 50.0,
                        LO_LIM := -50.0,
                        BIPOLAR := "TRUE",
                        OUT => "K1-334U":P);
   END_IF;
END_REGION

REGION Network 12: Останов сброса с рольганга
   RUNG wire#powerrail
      { S7_Templates := "SrcType := Int" } EQ_Contact(in1 := #BoardsInLayCounter, in2 := "ServDB".QPlanksInLayerBrak)
      { S7_Templates := "SrcType := Int" } NE_Contact(in1 := #BoardsInLayCounter, in2 := 0)
      S_SR(operand := #StopDropppingBoards, r1 := #ReviveSignal)
   END_RUNG
   // the same network as SCL:
   IF (#BoardsInLayCounter = "ServDB".QPlanksInLayerBrak) AND (#BoardsInLayCounter <> 0) THEN
       #StopDropppingBoards := TRUE;   // SR flip-flop
   END_IF;
   IF #ReviveSignal THEN #StopDropppingBoards := FALSE; END_IF;
END_REGION

REGION Network 13: Управление 332 транспортером
   RUNG wire#powerrail
      "BobDropper_CNTL_DB"(manCntl := wire#w1, bobFront := "DGI".BrakDroper_front, boardSig := "B22.0", fullLay := #StopDropppingBoards, CMD_ON =>)
      Contact( "ALG".Auto_defect )
      I_Contact( "ALG".Alarm_defect )
      Contact( "BobDropper_CNTL_DB".CMD_ON )
      Coil( "IM".M_332_Dump_lug_conv.OnCom )
   END_RUNG
   RUNG wire#powerrail
      Contact( "DGI".S79_4 )
      Contact( "ALG".Auto_defect )
   END_RUNG wire#w1
   // the same network as SCL:
   "BobDropper_CNTL_DB"(bobFront := "DGI".BrakDroper_front,   // "BobDropper_CNTL"
                        boardSig := "B22.0",
                        manCntl := "DGI".S79_4 AND "ALG".Auto_defect,
                        fullLay := #StopDropppingBoards,
                        ENO => #_w1);
   "IM".M_332_Dump_lug_conv.OnCom := #_w1 AND "ALG".Auto_defect AND NOT "ALG".Alarm_defect AND "BobDropper_CNTL_DB".CMD_ON;
END_REGION

REGION Network 14: М 332 Сброс с рольганга команды на движение
   RUNG wire#powerrail
      Contact( "ALG".Ready_defect )
      wire#w1
      Contact( "IM".M_332_Dump_lug_conv.onOutFWD )
      wire#w2
      "SolveSpeed"(GeneralSpeed := "VELOCITY".GeneralSpeed, MotorKoef := "VELOCITY".koef_M_332, Correction := 0.0, Ret_Val => "IM".M_332_Dump_lug_conv.setSpeedAU)
   END_RUNG
   RUNG wire#w2
      Not()
      { S7_GenerateENO := "TRUE" } Move(in := 0.0, out1 => "IM".M_332_Dump_lug_conv.setSpeedAU)
   END_RUNG
   RUNG wire#w1
      UNSCALE(IN := "IM".M_332_Dump_lug_conv.setSpeed, HI_LIM := 50.0, LO_LIM := -50.0, BIPOLAR := "TRUE", RET_VAL => #Sert, OUT => "K1-332U":P)
   END_RUNG
   // the same network as SCL:
   #_w1 := "ALG".Ready_defect AND "IM".M_332_Dump_lug_conv.onOutFWD;
   #_w2 := "ALG".Ready_defect;
   IF #_w1 THEN
       "IM".M_332_Dump_lug_conv.setSpeedAU := "SolveSpeed"(GeneralSpeed := "VELOCITY".GeneralSpeed,
                               MotorKoef := "VELOCITY".koef_M_332,
                               Correction := 0.0);
   END_IF;
   IF NOT #_w1 THEN "IM".M_332_Dump_lug_conv.setSpeedAU := 0.0; END_IF;
   IF #_w2 THEN
       #Sert := UNSCALE(IN := "IM".M_332_Dump_lug_conv.setSpeed,
                        HI_LIM := 50.0,
                        LO_LIM := -50.0,
                        BIPOLAR := "TRUE",
                        OUT => "K1-332U":P);
   END_IF;
END_REGION

REGION Network 15: Принудительно завершаем алгоритм сборки пакета (довод вил)
   RUNG wire#powerrail
      Contact( "ALG".ForceFinishPFMDefect )
      S_SR(operand := #ForcingPacket, r1 := wire#w1)
   END_RUNG
   RUNG wire#powerrail
      Contact( #ForcingLift )
   END_RUNG wire#w1
   // the same network as SCL:
   IF "ALG".ForceFinishPFMDefect THEN
       #ForcingPacket := TRUE;   // SR flip-flop
   END_IF;
   IF #ForcingLift THEN #ForcingPacket := FALSE; END_IF;
END_REGION

REGION Network 16: Форсирование сборки пакета ПФМ (лифт)
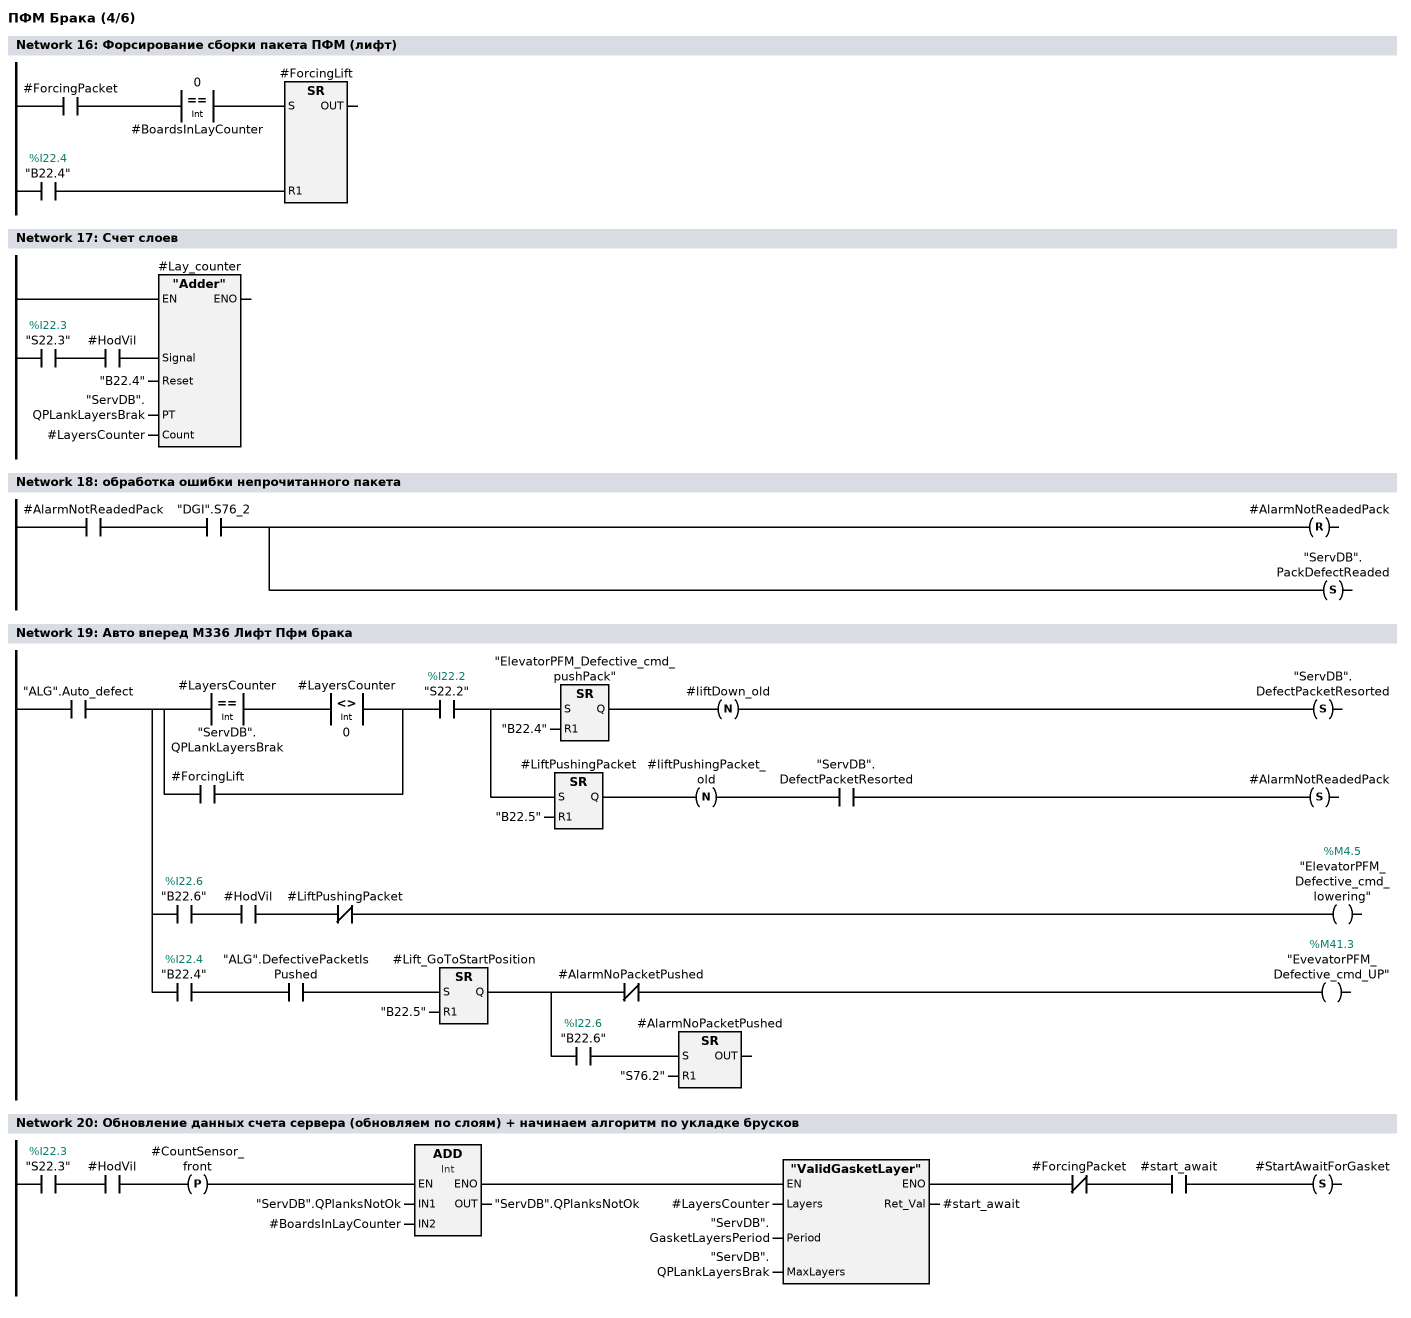
   RUNG wire#powerrail
      Contact( #ForcingPacket )
      { S7_Templates := "SrcType := Int" } EQ_Contact(in1 := 0, in2 := #BoardsInLayCounter)
      S_SR(operand := #ForcingLift, r1 := wire#w1)
   END_RUNG
   RUNG wire#powerrail
      Contact( "B22.4" )
   END_RUNG wire#w1
   // the same network as SCL:
   IF #ForcingPacket AND (0 = #BoardsInLayCounter) THEN
       #ForcingLift := TRUE;   // SR flip-flop
   END_IF;
   IF "B22.4" THEN #ForcingLift := FALSE; END_IF;
END_REGION

REGION Network 17: Счет слоев
   RUNG wire#powerrail
      #Lay_counter(Signal := wire#w1, Reset := "B22.4", PT := "ServDB".QPLankLayersBrak, Count := #LayersCounter)
   END_RUNG
   RUNG wire#powerrail
      Contact( "S22.3" )
      Contact( #HodVil )
   END_RUNG wire#w1
   // the same network as SCL:
   #Lay_counter(Signal := "S22.3" AND #HodVil,   // "Adder"
                Reset := "B22.4",
                PT := "ServDB".QPLankLayersBrak,
                Count := #LayersCounter);
END_REGION

REGION Network 18: обработка ошибки непрочитанного пакета
   RUNG wire#powerrail
      Contact( #AlarmNotReadedPack )
      Contact( "DGI".S76_2 )
      wire#w1
      R_Coil( #AlarmNotReadedPack )
   END_RUNG
   RUNG wire#w1
      S_Coil( "ServDB".PackDefectReaded )
   END_RUNG
   // the same network as SCL:
   #_w1 := #AlarmNotReadedPack AND "DGI".S76_2;
   IF #_w1 THEN
       #AlarmNotReadedPack := FALSE;
       "ServDB".PackDefectReaded := TRUE;
   END_IF;
END_REGION

REGION Network 19: Авто вперед М336 Лифт Пфм брака
   RUNG wire#powerrail
      Contact( "ALG".Auto_defect )
      wire#w1
      { S7_Templates := "SrcType := Int" } EQ_Contact(in1 := #LayersCounter, in2 := "ServDB".QPLankLayersBrak)
      { S7_Templates := "SrcType := Int" } NE_Contact(in1 := #LayersCounter, in2 := 0)
      wire#w2
      Contact( "S22.2" )
      wire#w3
      S_SR(operand := "ElevatorPFM_Defective_cmd_pushPack", r1 := "B22.4")
      N_Trig( #liftDown_old )
      S_Coil( "ServDB".DefectPacketResorted )
   END_RUNG
   RUNG wire#w1
      Contact( #ForcingLift )
   END_RUNG wire#w2
   RUNG wire#w3
      S_SR(operand := #LiftPushingPacket, r1 := "B22.5")
      N_Trig( #liftPushingPacket_old )
      Contact( "ServDB".DefectPacketResorted )
      S_Coil( #AlarmNotReadedPack )
   END_RUNG
   RUNG wire#w1
      Contact( "B22.6" )
      Contact( #HodVil )
      I_Contact( #LiftPushingPacket )
      Coil( "ElevatorPFM_Defective_cmd_lowering" )
   END_RUNG
   RUNG wire#w1
      Contact( "B22.4" )
      Contact( "ALG".DefectivePacketIsPushed )
      S_SR(operand := #Lift_GoToStartPosition, r1 := "B22.5")
      wire#w4
      I_Contact( #AlarmNoPacketPushed )
      Coil( "EvevatorPFM_Defective_cmd_UP" )
   END_RUNG
   RUNG wire#w4
      Contact( "B22.6" )
      S_SR(operand := #AlarmNoPacketPushed, r1 := "S76.2")
   END_RUNG
   // the same network as SCL:
   #_w1 := "ALG".Auto_defect AND (((#LayersCounter = "ServDB".QPLankLayersBrak) AND (#LayersCounter <> 0)) OR #ForcingLift) AND "S22.2";
   IF #_w1 THEN
       "ElevatorPFM_Defective_cmd_pushPack" := TRUE;   // SR flip-flop
   END_IF;
   IF "B22.4" THEN "ElevatorPFM_Defective_cmd_pushPack" := FALSE; END_IF;
   #_w2 := NOT "ElevatorPFM_Defective_cmd_pushPack" AND #liftDown_old;   // falling edge
   #liftDown_old := "ElevatorPFM_Defective_cmd_pushPack";
   IF #_w2 THEN "ServDB".DefectPacketResorted := TRUE; END_IF;
   IF #_w1 THEN
       #LiftPushingPacket := TRUE;   // SR flip-flop
   END_IF;
   IF "B22.5" THEN #LiftPushingPacket := FALSE; END_IF;
   #_w3 := NOT #LiftPushingPacket AND #liftPushingPacket_old;   // falling edge
   #liftPushingPacket_old := #LiftPushingPacket;
   IF #_w3 AND "ServDB".DefectPacketResorted THEN #AlarmNotReadedPack := TRUE; END_IF;
   "ElevatorPFM_Defective_cmd_lowering" := "ALG".Auto_defect AND "B22.6" AND #HodVil AND NOT #LiftPushingPacket;
   IF "ALG".Auto_defect AND "B22.4" AND "ALG".DefectivePacketIsPushed THEN
       #Lift_GoToStartPosition := TRUE;   // SR flip-flop
   END_IF;
   IF "B22.5" THEN #Lift_GoToStartPosition := FALSE; END_IF;
   "EvevatorPFM_Defective_cmd_UP" := #Lift_GoToStartPosition AND NOT #AlarmNoPacketPushed;
   IF #Lift_GoToStartPosition AND "B22.6" THEN
       #AlarmNoPacketPushed := TRUE;   // SR flip-flop
   END_IF;
   IF "S76.2" THEN #AlarmNoPacketPushed := FALSE; END_IF;
END_REGION

REGION Network 20: Обновление данных счета сервера (обновляем по слоям) + начинаем алгоритм по укладке брусков
   RUNG wire#powerrail
      Contact( "S22.3" )
      Contact( #HodVil )
      P_Trig( #CountSensor_front )
      { S7_Templates := "SrcType := Int"; S7_GenerateENO := "TRUE" } Add(in1 := "ServDB".QPlanksNotOk, in2 := #BoardsInLayCounter, out => "ServDB".QPlanksNotOk)
      "ValidGasketLayer"(Layers := #LayersCounter, Period := "ServDB".GasketLayersPeriod, MaxLayers := "ServDB".QPLankLayersBrak, Ret_Val => #start_await)
      I_Contact( #ForcingPacket )
      Contact( #start_await )
      S_Coil( #StartAwaitForGasket )
   END_RUNG
   // the same network as SCL:
   // ENO of a box is taken as its EN; it also drops when the box reports an error
   #_w1 := "S22.3" AND #HodVil;
   #_w2 := #_w1 AND NOT #CountSensor_front;   // rising edge
   #CountSensor_front := #_w1;
   IF #_w2 THEN "ServDB".QPlanksNotOk := "ServDB".QPlanksNotOk + #BoardsInLayCounter; END_IF;
   #start_await := "ValidGasketLayer"(EN := #_w2,
                           Layers := #LayersCounter,
                           Period := "ServDB".GasketLayersPeriod,
                           MaxLayers := "ServDB".QPLankLayersBrak,
                           ENO => #_w3);
   IF #_w3 AND NOT #ForcingPacket AND #start_await THEN #StartAwaitForGasket := TRUE; END_IF;
END_REGION

REGION Network 21: Логика ожидания уложенных прокладок на пакет Брака
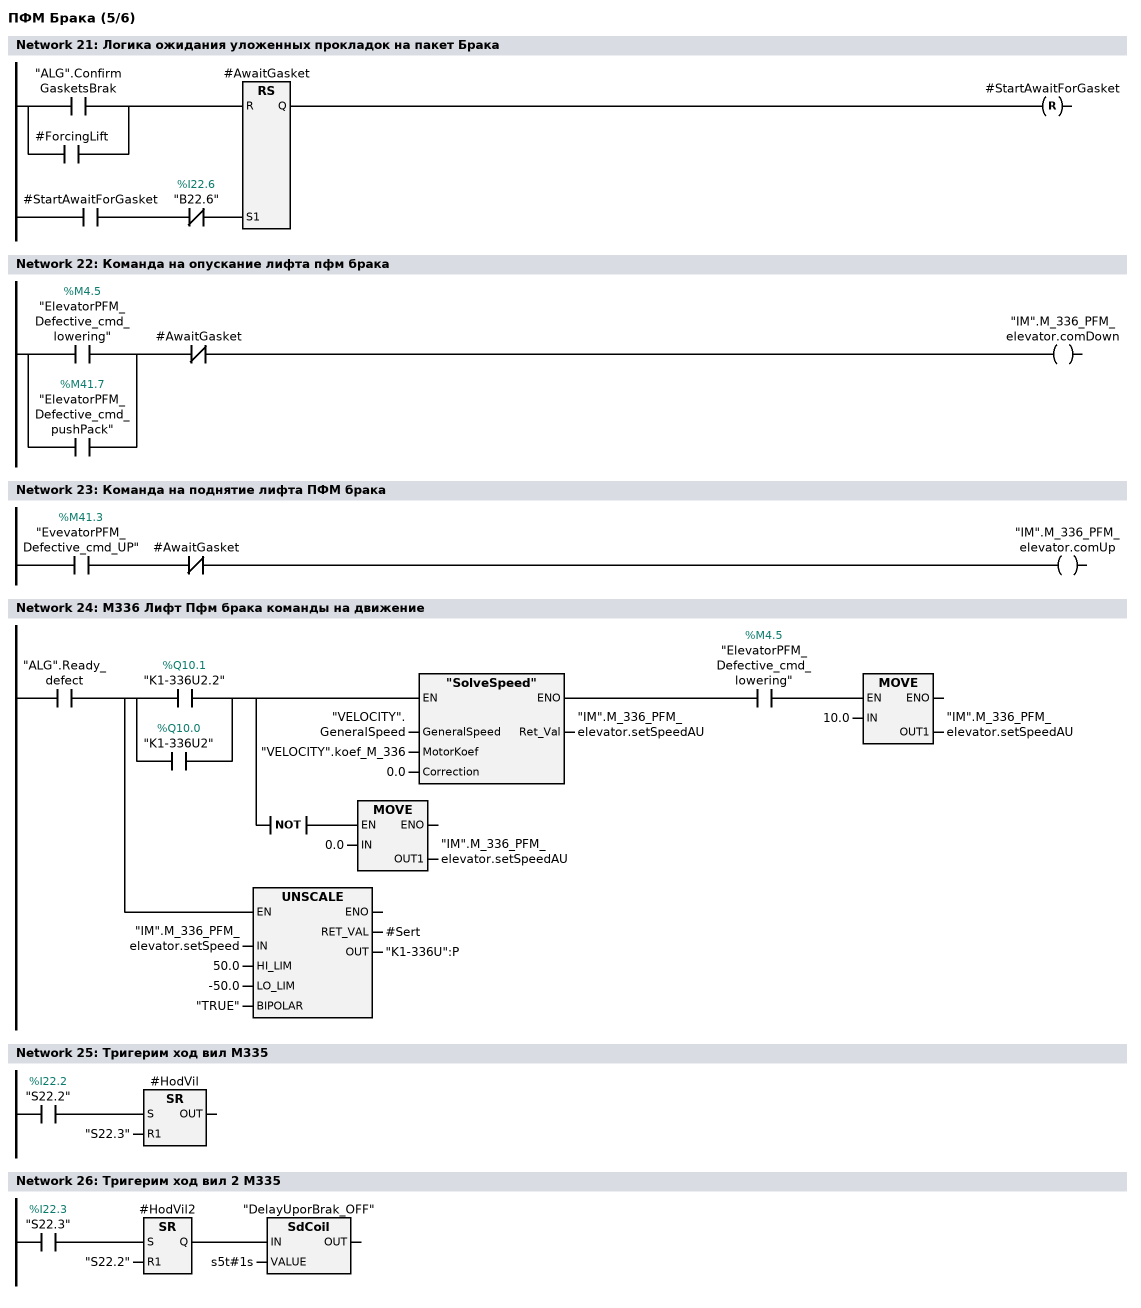
   RUNG wire#powerrail
      Contact( "ALG".ConfirmGasketsBrak )
      wire#w1
      S_RS(operand := #AwaitGasket, s1 := wire#w2)
      R_Coil( #StartAwaitForGasket )
   END_RUNG
   RUNG wire#powerrail
      Contact( #ForcingLift )
   END_RUNG wire#w1
   RUNG wire#powerrail
      Contact( #StartAwaitForGasket )
      I_Contact( "B22.6" )
   END_RUNG wire#w2
   // the same network as SCL:
   IF "ALG".ConfirmGasketsBrak OR #ForcingLift THEN
       #AwaitGasket := FALSE;   // RS flip-flop
   END_IF;
   IF #StartAwaitForGasket AND NOT "B22.6" THEN #AwaitGasket := TRUE; END_IF;
   IF #AwaitGasket THEN #StartAwaitForGasket := FALSE; END_IF;
END_REGION

REGION Network 22: Команда на опускание лифта пфм брака
   RUNG wire#powerrail
      Contact( "ElevatorPFM_Defective_cmd_lowering" )
      wire#w1
      I_Contact( #AwaitGasket )
      Coil( "IM".M_336_PFM_elevator.comDown )
   END_RUNG
   RUNG wire#powerrail
      Contact( "ElevatorPFM_Defective_cmd_pushPack" )
   END_RUNG wire#w1
   // the same network as SCL:
   "IM".M_336_PFM_elevator.comDown := ("ElevatorPFM_Defective_cmd_lowering" OR "ElevatorPFM_Defective_cmd_pushPack") AND NOT #AwaitGasket;
END_REGION

REGION Network 23: Команда на поднятие лифта ПФМ брака
   RUNG wire#powerrail
      Contact( "EvevatorPFM_Defective_cmd_UP" )
      I_Contact( #AwaitGasket )
      Coil( "IM".M_336_PFM_elevator.comUp )
   END_RUNG
   // the same network as SCL:
   "IM".M_336_PFM_elevator.comUp := "EvevatorPFM_Defective_cmd_UP" AND NOT #AwaitGasket;
END_REGION

REGION Network 24: М336 Лифт Пфм брака команды на движение
   RUNG wire#powerrail
      Contact( "ALG".Ready_defect )
      wire#w1
      Contact( "K1-336U2.2" )
      wire#w2
      "SolveSpeed"(GeneralSpeed := "VELOCITY".GeneralSpeed, MotorKoef := "VELOCITY".koef_M_336, Correction := 0.0, Ret_Val => "IM".M_336_PFM_elevator.setSpeedAU)
      Contact( "ElevatorPFM_Defective_cmd_lowering" )
      { S7_GenerateENO := "TRUE" } Move(in := 10.0, out1 => "IM".M_336_PFM_elevator.setSpeedAU)
   END_RUNG
   RUNG wire#w1
      Contact( "K1-336U2" )
   END_RUNG wire#w2
   RUNG wire#w2
      Not()
      { S7_GenerateENO := "TRUE" } Move(in := 0.0, out1 => "IM".M_336_PFM_elevator.setSpeedAU)
   END_RUNG
   RUNG wire#w1
      UNSCALE(IN := "IM".M_336_PFM_elevator.setSpeed, HI_LIM := 50.0, LO_LIM := -50.0, BIPOLAR := "TRUE", RET_VAL => #Sert, OUT => "K1-336U":P)
   END_RUNG
   // the same network as SCL:
   #_w1 := "ALG".Ready_defect AND ("K1-336U2.2" OR "K1-336U2");
   #_w3 := "ALG".Ready_defect;
   "IM".M_336_PFM_elevator.setSpeedAU := "SolveSpeed"(EN := #_w1,
                           GeneralSpeed := "VELOCITY".GeneralSpeed,
                           MotorKoef := "VELOCITY".koef_M_336,
                           Correction := 0.0,
                           ENO => #_w2);
   IF #_w2 AND "ElevatorPFM_Defective_cmd_lowering" THEN "IM".M_336_PFM_elevator.setSpeedAU := 10.0; END_IF;
   IF NOT #_w1 THEN "IM".M_336_PFM_elevator.setSpeedAU := 0.0; END_IF;
   IF #_w3 THEN
       #Sert := UNSCALE(IN := "IM".M_336_PFM_elevator.setSpeed,
                        HI_LIM := 50.0,
                        LO_LIM := -50.0,
                        BIPOLAR := "TRUE",
                        OUT => "K1-336U":P);
   END_IF;
END_REGION

REGION Network 25: Тригерим ход вил М335
   RUNG wire#powerrail
      Contact( "S22.2" )
      S_SR(operand := #HodVil, r1 := "S22.3")
   END_RUNG
   // the same network as SCL:
   IF "S22.2" THEN
       #HodVil := TRUE;   // SR flip-flop
   END_IF;
   IF "S22.3" THEN #HodVil := FALSE; END_IF;
END_REGION

REGION Network 26: Тригерим ход вил 2 М335
   // no SCL statement known for SdCoil: written as a call
   IF "S22.3" THEN
       #HodVil2 := TRUE;   // SR flip-flop
   END_IF;
   IF "S22.2" THEN #HodVil2 := FALSE; END_IF;
   SdCoil(in := #HodVil2, value := s5t#1s, operand := "DelayUporBrak_OFF");
END_REGION

REGION Network 27: авария убрать лишнюю доску с ПФМ брака
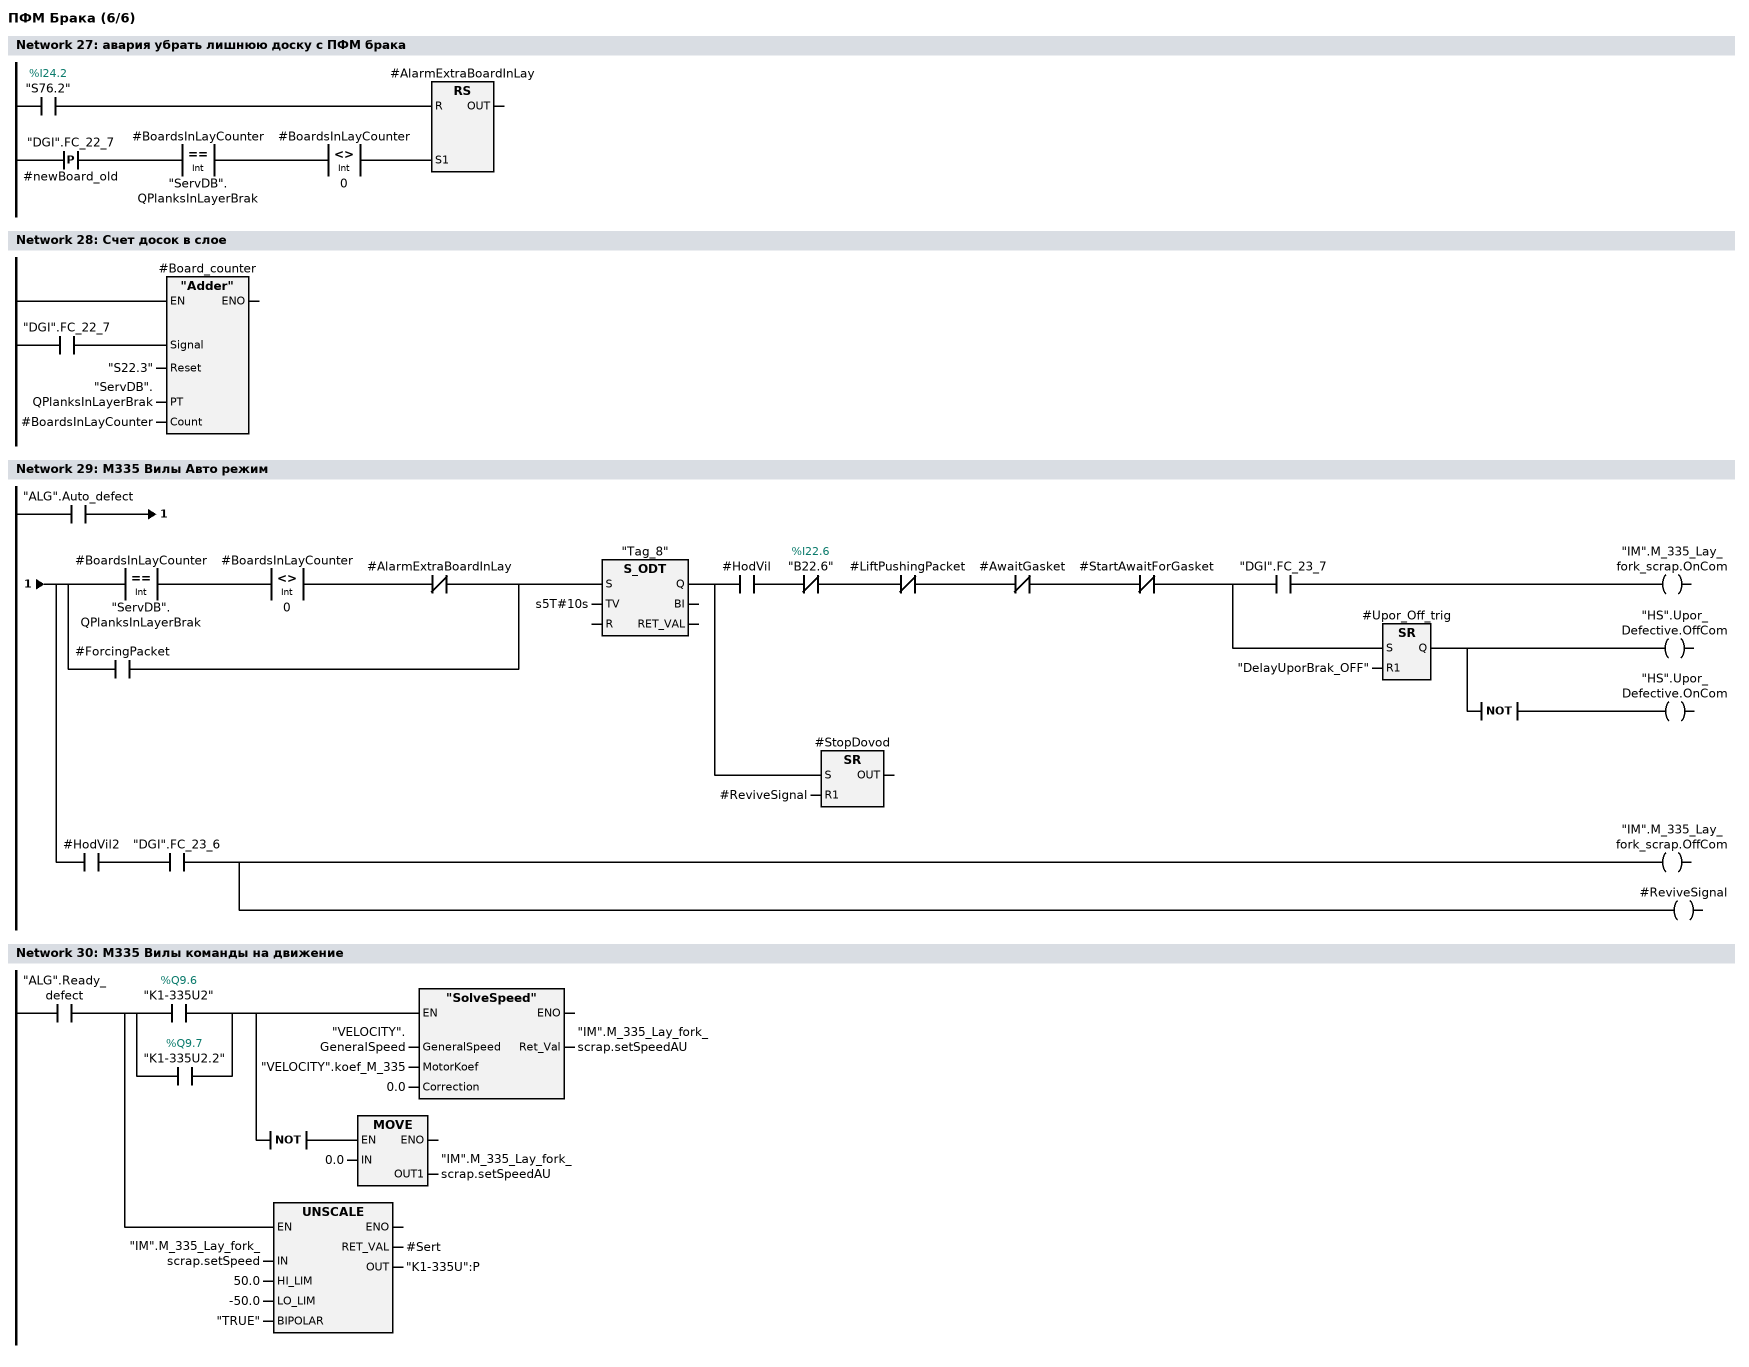
   RUNG wire#powerrail
      Contact( "S76.2" )
      S_RS(operand := #AlarmExtraBoardInLay, s1 := wire#w1)
   END_RUNG
   RUNG wire#powerrail
      P_Contact(operand := "DGI".FC_22_7, bit := #newBoard_old)
      { S7_Templates := "SrcType := Int" } EQ_Contact(in1 := #BoardsInLayCounter, in2 := "ServDB".QPlanksInLayerBrak)
      { S7_Templates := "SrcType := Int" } NE_Contact(in1 := #BoardsInLayCounter, in2 := 0)
   END_RUNG wire#w1
   // the same network as SCL:
   #_w1 := "DGI".FC_22_7 AND NOT #newBoard_old;   // rising edge of "DGI".FC_22_7
   #newBoard_old := "DGI".FC_22_7;
   IF "S76.2" THEN
       #AlarmExtraBoardInLay := FALSE;   // RS flip-flop
   END_IF;
   IF #_w1 AND (#BoardsInLayCounter = "ServDB".QPlanksInLayerBrak) AND (#BoardsInLayCounter <> 0) THEN
       #AlarmExtraBoardInLay := TRUE;
   END_IF;
END_REGION

REGION Network 28: Счет досок в слое
   RUNG wire#powerrail
      #Board_counter(Signal := wire#w1, Reset := "S22.3", PT := "ServDB".QPlanksInLayerBrak, Count := #BoardsInLayCounter)
   END_RUNG
   RUNG wire#powerrail
      Contact( "DGI".FC_22_7 )
   END_RUNG wire#w1
   // the same network as SCL:
   #Board_counter(Signal := "DGI".FC_22_7,   // "Adder"
                  Reset := "S22.3",
                  PT := "ServDB".QPlanksInLayerBrak,
                  Count := #BoardsInLayCounter);
END_REGION

REGION Network 29: М335 Вилы Авто режим
   RUNG wire#powerrail
      Contact( "ALG".Auto_defect )
      wire#w1
      { S7_Templates := "SrcType := Int" } EQ_Contact(in1 := #BoardsInLayCounter, in2 := "ServDB".QPlanksInLayerBrak)
      { S7_Templates := "SrcType := Int" } NE_Contact(in1 := #BoardsInLayCounter, in2 := 0)
      I_Contact( #AlarmExtraBoardInLay )
      wire#w2
      S_ODT(T_NO := "Tag_8", TV := s5T#10s, R :=, BI =>, RET_VAL =>)
      wire#w3
      Contact( #HodVil )
      I_Contact( "B22.6" )
      I_Contact( #LiftPushingPacket )
      I_Contact( #AwaitGasket )
      I_Contact( #StartAwaitForGasket )
      wire#w4
      Contact( "DGI".FC_23_7 )
      Coil( "IM".M_335_Lay_fork_scrap.OnCom )
   END_RUNG
   RUNG wire#w1
      Contact( #ForcingPacket )
   END_RUNG wire#w2
   RUNG wire#w4
      S_SR(operand := #Upor_Off_trig, r1 := "DelayUporBrak_OFF")
      wire#w5
      Coil( "HS".Upor_Defective.OffCom )
   END_RUNG
   RUNG wire#w5
      Not()
      Coil( "HS".Upor_Defective.OnCom )
   END_RUNG
   RUNG wire#w3
      S_SR(operand := #StopDovod, r1 := #ReviveSignal)
   END_RUNG
   RUNG wire#w1
      Contact( #HodVil2 )
      Contact( "DGI".FC_23_6 )
      wire#w6
      Coil( "IM".M_335_Lay_fork_scrap.OffCom )
   END_RUNG
   RUNG wire#w6
      Coil( #ReviveSignal )
   END_RUNG
   // the same network as SCL:
   #_w2 := "ALG".Auto_defect;
   #_s5time1 := S_ODT(T_NO := "Tag_8",
                      S := "ALG".Auto_defect AND (((#BoardsInLayCounter = "ServDB".QPlanksInLayerBrak) AND (#BoardsInLayCounter <> 0) AND NOT #AlarmExtraBoardInLay) OR #ForcingPacket),
                      TV := s5T#10s,
                      Q => #_w1);
   #_w3 := #_w1 AND #HodVil AND NOT "B22.6" AND NOT #LiftPushingPacket AND NOT #AwaitGasket AND NOT #StartAwaitForGasket;
   "IM".M_335_Lay_fork_scrap.OnCom := #_w3 AND "DGI".FC_23_7;
   IF #_w3 THEN
       #Upor_Off_trig := TRUE;   // SR flip-flop
   END_IF;
   IF "DelayUporBrak_OFF" THEN #Upor_Off_trig := FALSE; END_IF;
   "HS".Upor_Defective.OffCom := #Upor_Off_trig;
   "HS".Upor_Defective.OnCom := NOT #Upor_Off_trig;
   IF #_w1 THEN
       #StopDovod := TRUE;   // SR flip-flop
   END_IF;
   IF #ReviveSignal THEN #StopDovod := FALSE; END_IF;
   "IM".M_335_Lay_fork_scrap.OffCom := #_w2 AND #HodVil2 AND "DGI".FC_23_6;
   #ReviveSignal := "IM".M_335_Lay_fork_scrap.OffCom;
END_REGION

REGION Network 30: М335 Вилы команды на движение
   RUNG wire#powerrail
      Contact( "ALG".Ready_defect )
      wire#w1
      Contact( "K1-335U2" )
      wire#w2
      "SolveSpeed"(GeneralSpeed := "VELOCITY".GeneralSpeed, MotorKoef := "VELOCITY".koef_M_335, Correction := 0.0, Ret_Val => "IM".M_335_Lay_fork_scrap.setSpeedAU)
   END_RUNG
   RUNG wire#w1
      Contact( "K1-335U2.2" )
   END_RUNG wire#w2
   RUNG wire#w2
      Not()
      { S7_GenerateENO := "TRUE" } Move(in := 0.0, out1 => "IM".M_335_Lay_fork_scrap.setSpeedAU)
   END_RUNG
   RUNG wire#w1
      UNSCALE(IN := "IM".M_335_Lay_fork_scrap.setSpeed, HI_LIM := 50.0, LO_LIM := -50.0, BIPOLAR := "TRUE", RET_VAL => #Sert, OUT => "K1-335U":P)
   END_RUNG
   // the same network as SCL:
   #_w1 := "ALG".Ready_defect AND ("K1-335U2" OR "K1-335U2.2");
   #_w2 := "ALG".Ready_defect;
   IF #_w1 THEN
       "IM".M_335_Lay_fork_scrap.setSpeedAU := "SolveSpeed"(GeneralSpeed := "VELOCITY".GeneralSpeed,
                               MotorKoef := "VELOCITY".koef_M_335,
                               Correction := 0.0);
   END_IF;
   IF NOT #_w1 THEN "IM".M_335_Lay_fork_scrap.setSpeedAU := 0.0; END_IF;
   IF #_w2 THEN
       #Sert := UNSCALE(IN := "IM".M_335_Lay_fork_scrap.setSpeed,
                        HI_LIM := 50.0,
                        LO_LIM := -50.0,
                        BIPOLAR := "TRUE",
                        OUT => "K1-335U":P);
   END_IF;
END_REGION
END_FUNCTION_BLOCK

FUNCTION_BLOCK "BobDropper_CNTL"
{ S7_Optimized_Access := 'FALSE' }
AUTHOR : Aspir
VERSION : 0.1
   VAR_INPUT 
      bobFront { ExternalAccessible := 'False'; ExternalVisible := 'False'; ExternalWritable := 'False'} : Bool;
      boardSig : Bool;   // сигнал наличия доски
      manCntl : Bool;   // ручной выгон (1 прокрут)
      fullLay : Bool;   // полный слой собран
   END_VAR

   VAR_OUTPUT 
      CMD_ON : Bool;   // команда на движение сброса с бобышек
   END_VAR

   VAR 
      DropTask : Bool;   // задание на выгон доски целиком
      ShiftTask : Bool;   // задание на сдвиг доски
      Shifted : Bool;   // сдвинут на бобыльку
      Vibrator : Bool;
      DropTask_old : Bool;
      ValidBoard_timer {InstructionName := 'TON'; LibVersion := '1.0'; S7_SetPoint := 'False'} : TON;   // таймер наличия доски
   END_VAR

   VAR CONSTANT 
      filterDelay : Time := T#100ms;
   END_VAR


BEGIN
	//Фильтр наличия доски
	//
	#ValidBoard_timer(IN:=#boardSig,
	                  PT:=#filterDelay);
	
	// задание на сброс доски (2 прокрута)
	//
	#DropTask := (#DropTask OR (#ValidBoard_timer.Q OR #manCntl)) AND NOT (#fullLay OR #Vibrator AND #bobFront); // задание на прокрут полный
	
	// помогает проехать две бобышки вместо одной
	// инвертирует только при 
	#Vibrator := (#Vibrator XOR (#DropTask AND #bobFront)) AND NOT (#DropTask AND NOT #DropTask_old);
	
	// Задание на сдвиг доски на одну бобышку
	// 
	#Shifted := (#Shifted OR #bobFront AND #ShiftTask) AND NOT #DropTask; // запоминаем что мы сдвинуты
	#ShiftTask := (#ShiftTask OR #ValidBoard_timer.Q AND #fullLay AND NOT #Shifted) AND NOT (#bobFront); //задание на сдвиг на одну бобышку
	
	
	// Команды и сигналы на выход
	// 
	#CMD_ON := #ShiftTask OR #DropTask;
	
	// ловим фронты
	// 
	#DropTask_old := #DropTask;
END_FUNCTION_BLOCK

FUNCTION_BLOCK "Adder"
{ S7_Optimized_Access := 'FALSE' }
VERSION : 0.1
   VAR_INPUT 
      Signal : Bool;   // входной сигнал
      Reset : Bool;   // сброс счетчика
      PT : Int;   // Пресет счетчика
   END_VAR

   VAR_IN_OUT 
      Count : Int;
   END_VAR

   VAR 
      Signal_old : Bool;
   END_VAR


BEGIN
	IF (#Signal AND NOT #Signal_old AND #Count < #PT ) THEN
	    #Count := #Count + 1;
	END_IF;
	
	IF (#Reset) THEN
	    #Count := 0;
	END_IF;
	
	#Signal_old := #Signal;
END_FUNCTION_BLOCK

FUNCTION "ValidGasketLayer" : Bool
{ S7_Optimized_Access := 'FALSE' }
VERSION : 0.1
   VAR_INPUT 
      Layers : Int;
      Period : Int;
      MaxLayers : Int;
   END_VAR


BEGIN
	IF (#Period <> 0) THEN
	    #ValidGasketLayer := (#Layers MOD #Period = 0) AND NOT (#Layers = 0 OR #Layers = #MaxLayers);
	ELSE
	    #ValidGasketLayer := FALSE;
	END_IF;
	
END_FUNCTION

FUNCTION_BLOCK "Подача прокладки"   // FB6, LAD
VERSION : 0.1
// Подача прокладки
// stored: AutoNumber true, IsIECCheckEnabled false, UDAEnableTagReadback false
   VAR DB_SPECIFIC
      "TrigS84.4/S79.1" : Bool;
      Trig315 : Bool;
   END_VAR
   VAR_TEMP   // added for the SCL form of the ladder/FBD networks
      _w1 : Bool;
      _s5time1 : S5Time;
      _w2 : Bool;
      _w3 : Bool;
      _s5time2 : S5Time;
   END_VAR
BEGIN

REGION Network 1: Готовность
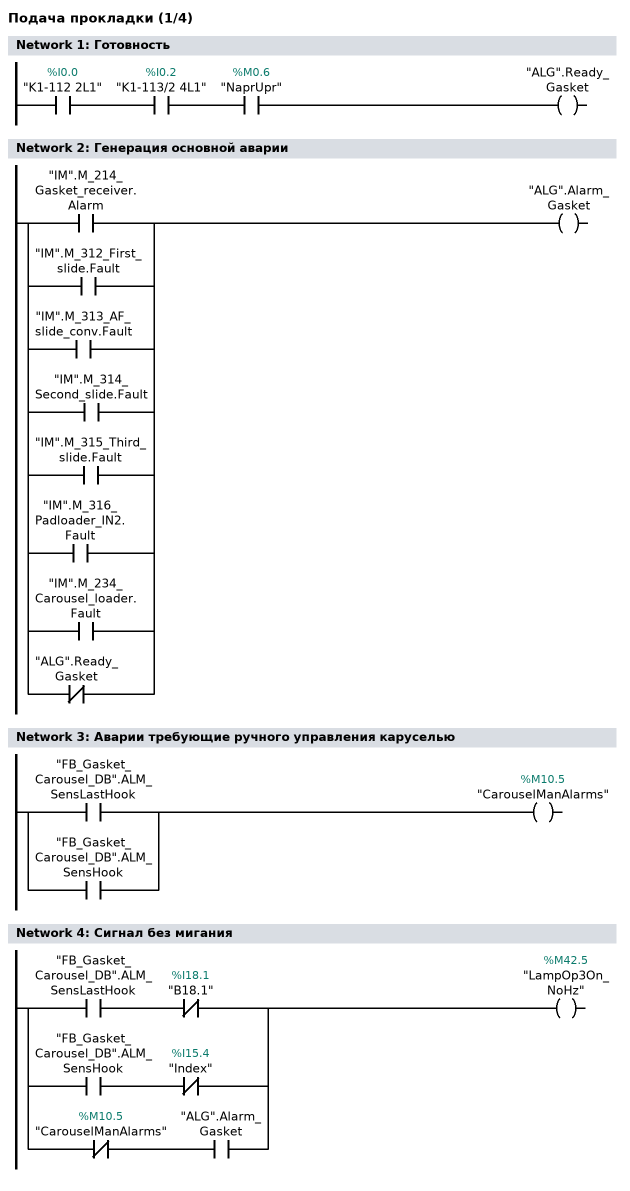
   RUNG wire#powerrail
      Contact( "K1-112 2L1" )
      Contact( "K1-113/2 4L1" )
      Contact( "NaprUpr" )
      Coil( "ALG".Ready_Gasket )
   END_RUNG
   // the same network as SCL:
   "ALG".Ready_Gasket := "K1-112 2L1" AND "K1-113/2 4L1" AND "NaprUpr";
END_REGION

REGION Network 2: Генерация основной аварии
   RUNG wire#powerrail
      Contact( "IM".M_214_Gasket_receiver.Alarm )
      wire#w1
      Coil( "ALG".Alarm_Gasket )
   END_RUNG
   RUNG wire#powerrail
      Contact( "IM".M_312_First_slide.Fault )
   END_RUNG wire#w1
   RUNG wire#powerrail
      Contact( "IM".M_313_AF_slide_conv.Fault )
   END_RUNG wire#w1
   RUNG wire#powerrail
      Contact( "IM".M_314_Second_slide.Fault )
   END_RUNG wire#w1
   RUNG wire#powerrail
      Contact( "IM".M_315_Third_slide.Fault )
   END_RUNG wire#w1
   RUNG wire#powerrail
      Contact( "IM".M_316_Padloader_IN2.Fault )
   END_RUNG wire#w1
   RUNG wire#powerrail
      Contact( "IM".M_234_Carousel_loader.Fault )
   END_RUNG wire#w1
   RUNG wire#powerrail
      I_Contact( "ALG".Ready_Gasket )
   END_RUNG wire#w1
   // the same network as SCL:
   "ALG".Alarm_Gasket := "IM".M_214_Gasket_receiver.Alarm OR "IM".M_312_First_slide.Fault OR "IM".M_313_AF_slide_conv.Fault OR "IM".M_314_Second_slide.Fault OR "IM".M_315_Third_slide.Fault OR "IM".M_316_Padloader_IN2.Fault OR "IM".M_234_Carousel_loader.Fault OR NOT "ALG".Ready_Gasket;
END_REGION

REGION Network 3: Аварии требующие ручного управления каруселью
   RUNG wire#powerrail
      Contact( "FB_Gasket_Carousel_DB".ALM_SensLastHook )
      wire#w1
      Coil( "CarouselManAlarms" )
   END_RUNG
   RUNG wire#powerrail
      Contact( "FB_Gasket_Carousel_DB".ALM_SensHook )
   END_RUNG wire#w1
   // the same network as SCL:
   "CarouselManAlarms" := "FB_Gasket_Carousel_DB".ALM_SensLastHook OR "FB_Gasket_Carousel_DB".ALM_SensHook;
END_REGION

REGION Network 4: Сигнал без мигания
   RUNG wire#powerrail
      Contact( "FB_Gasket_Carousel_DB".ALM_SensLastHook )
      I_Contact( "B18.1" )
      wire#w1
      Coil( "LampOp3On_NoHz" )
   END_RUNG
   RUNG wire#powerrail
      Contact( "FB_Gasket_Carousel_DB".ALM_SensHook )
      I_Contact( "Index" )
   END_RUNG wire#w1
   RUNG wire#powerrail
      I_Contact( "CarouselManAlarms" )
      Contact( "ALG".Alarm_Gasket )
   END_RUNG wire#w1
   // the same network as SCL:
   "LampOp3On_NoHz" := ("FB_Gasket_Carousel_DB".ALM_SensLastHook AND NOT "B18.1") OR ("FB_Gasket_Carousel_DB".ALM_SensHook AND NOT "Index") OR (NOT "CarouselManAlarms" AND "ALG".Alarm_Gasket);
END_REGION

REGION Network 5: Сигнал об авариях с миганием
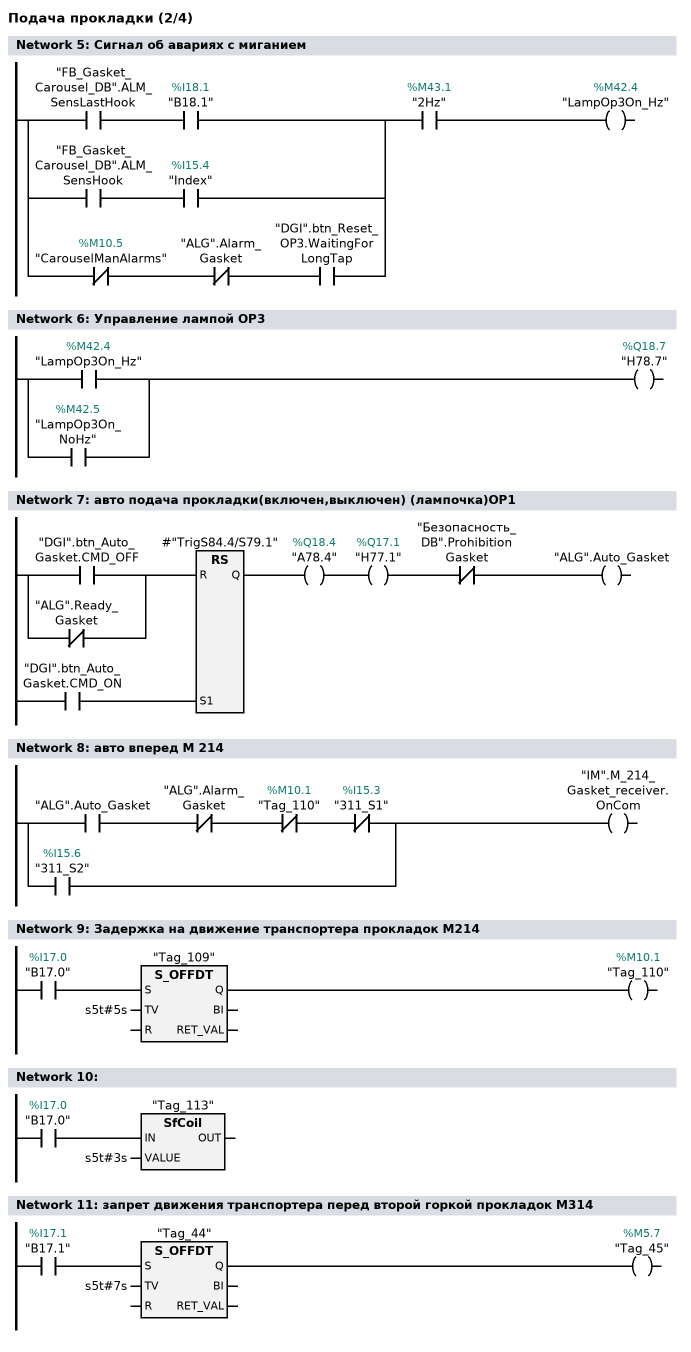
   RUNG wire#powerrail
      Contact( "FB_Gasket_Carousel_DB".ALM_SensLastHook )
      Contact( "B18.1" )
      wire#w1
      Contact( "2Hz" )
      Coil( "LampOp3On_Hz" )
   END_RUNG
   RUNG wire#powerrail
      Contact( "FB_Gasket_Carousel_DB".ALM_SensHook )
      Contact( "Index" )
   END_RUNG wire#w1
   RUNG wire#powerrail
      I_Contact( "CarouselManAlarms" )
      I_Contact( "ALG".Alarm_Gasket )
      Contact( "DGI".btn_Reset_OP3.WaitingForLongTap )
   END_RUNG wire#w1
   // the same network as SCL:
   "LampOp3On_Hz" := (("FB_Gasket_Carousel_DB".ALM_SensLastHook AND "B18.1") OR ("FB_Gasket_Carousel_DB".ALM_SensHook AND "Index") OR (NOT "CarouselManAlarms" AND NOT "ALG".Alarm_Gasket AND "DGI".btn_Reset_OP3.WaitingForLongTap)) AND "2Hz";
END_REGION

REGION Network 6: Управление лампой OP3
   RUNG wire#powerrail
      Contact( "LampOp3On_Hz" )
      wire#w1
      Coil( "H78.7" )
   END_RUNG
   RUNG wire#powerrail
      Contact( "LampOp3On_NoHz" )
   END_RUNG wire#w1
   // the same network as SCL:
   "H78.7" := "LampOp3On_Hz" OR "LampOp3On_NoHz";
END_REGION

REGION Network 7: авто подача прокладки(включен,выключен) (лампочка)ОР1
   RUNG wire#powerrail
      Contact( "DGI".btn_Auto_Gasket.CMD_OFF )
      wire#w1
      S_RS(operand := #"TrigS84.4/S79.1", s1 := wire#w2)
      Coil( "A78.4" )
      Coil( "H77.1" )
      I_Contact( "Безопасность_DB".ProhibitionGasket )
      Coil( "ALG".Auto_Gasket )
   END_RUNG
   RUNG wire#powerrail
      I_Contact( "ALG".Ready_Gasket )
   END_RUNG wire#w1
   RUNG wire#powerrail
      Contact( "DGI".btn_Auto_Gasket.CMD_ON )
   END_RUNG wire#w2
   // the same network as SCL:
   IF "DGI".btn_Auto_Gasket.CMD_OFF OR NOT "ALG".Ready_Gasket THEN
       #"TrigS84.4/S79.1" := FALSE;   // RS flip-flop
   END_IF;
   IF "DGI".btn_Auto_Gasket.CMD_ON THEN #"TrigS84.4/S79.1" := TRUE; END_IF;
   "A78.4" := #"TrigS84.4/S79.1";
   "H77.1" := #"TrigS84.4/S79.1";
   "ALG".Auto_Gasket := #"TrigS84.4/S79.1" AND NOT "Безопасность_DB".ProhibitionGasket;
END_REGION

REGION Network 8: авто вперед M 214
   RUNG wire#powerrail
      Contact( "ALG".Auto_Gasket )
      I_Contact( "ALG".Alarm_Gasket )
      I_Contact( "Tag_110" )
      I_Contact( "311_S1" )
      wire#w1
      Coil( "IM".M_214_Gasket_receiver.OnCom )
   END_RUNG
   RUNG wire#powerrail
      Contact( "311_S2" )
   END_RUNG wire#w1
   // the same network as SCL:
   "IM".M_214_Gasket_receiver.OnCom := ("ALG".Auto_Gasket AND NOT "ALG".Alarm_Gasket AND NOT "Tag_110" AND NOT "311_S1") OR "311_S2";
END_REGION

REGION Network 9: Задержка на движение транспортера прокладок М214
   RUNG wire#powerrail
      Contact( "B17.0" )
      S_OFFDT(T_NO := "Tag_109", TV := s5t#5s, R :=, BI =>, RET_VAL =>)
      Coil( "Tag_110" )
   END_RUNG
   // the same network as SCL:
   #_s5time1 := S_OFFDT(T_NO := "Tag_109", S := "B17.0", TV := s5t#5s, Q => #_w1);
   "Tag_110" := #_w1;
END_REGION

REGION Network 10
   // no SCL statement known for SfCoil: written as a call
   SfCoil(in := "B17.0", value := s5t#3s, operand := "Tag_113");
END_REGION

REGION Network 11: запрет движения транспортера перед второй горкой прокладок М314
   RUNG wire#powerrail
      Contact( "B17.1" )
      S_OFFDT(T_NO := "Tag_44", TV := s5t#7s, R :=, BI =>, RET_VAL =>)
      Coil( "Tag_45" )
   END_RUNG
   // the same network as SCL:
   #_s5time1 := S_OFFDT(T_NO := "Tag_44", S := "B17.1", TV := s5t#7s, Q => #_w1);
   "Tag_45" := #_w1;
END_REGION

REGION Network 12: Авто вперед команда подачи прокладок до горок
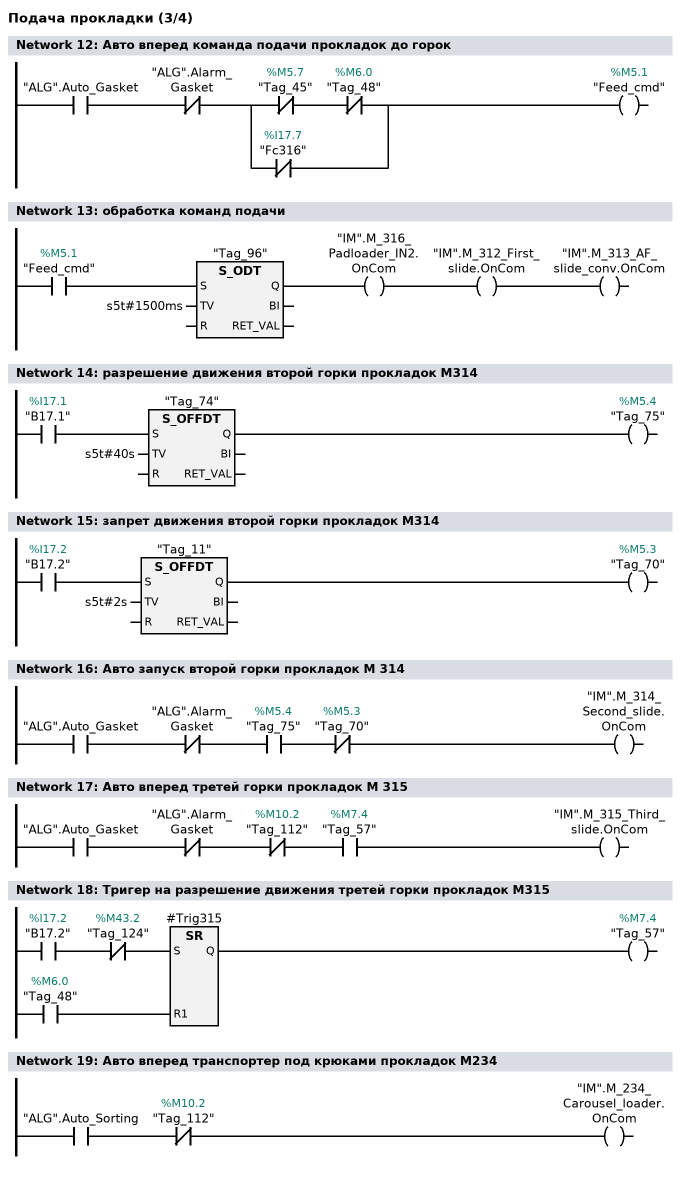
   RUNG wire#powerrail
      Contact( "ALG".Auto_Gasket )
      I_Contact( "ALG".Alarm_Gasket )
      wire#w1
      I_Contact( "Tag_45" )
      I_Contact( "Tag_48" )
      wire#w2
      Coil( "Feed_cmd" )
   END_RUNG
   RUNG wire#w1
      I_Contact( "Fc316" )
   END_RUNG wire#w2
   // the same network as SCL:
   "Feed_cmd" := "ALG".Auto_Gasket AND NOT "ALG".Alarm_Gasket AND ((NOT "Tag_45" AND NOT "Tag_48") OR NOT "Fc316");
END_REGION

REGION Network 13: обработка команд подачи
   RUNG wire#powerrail
      Contact( "Feed_cmd" )
      S_ODT(T_NO := "Tag_96", TV := s5t#1500ms, R :=, BI =>, RET_VAL =>)
      Coil( "IM".M_316_Padloader_IN2.OnCom )
      Coil( "IM".M_312_First_slide.OnCom )
      Coil( "IM".M_313_AF_slide_conv.OnCom )
   END_RUNG
   // the same network as SCL:
   #_s5time1 := S_ODT(T_NO := "Tag_96", S := "Feed_cmd", TV := s5t#1500ms, Q => #_w1);
   "IM".M_316_Padloader_IN2.OnCom := #_w1;
   "IM".M_312_First_slide.OnCom := #_w1;
   "IM".M_313_AF_slide_conv.OnCom := #_w1;
END_REGION

REGION Network 14: разрешение движения второй горки прокладок М314
   RUNG wire#powerrail
      Contact( "B17.1" )
      S_OFFDT(T_NO := "Tag_74", TV := s5t#40s, R :=, BI =>, RET_VAL =>)
      Coil( "Tag_75" )
   END_RUNG
   // the same network as SCL:
   #_s5time1 := S_OFFDT(T_NO := "Tag_74", S := "B17.1", TV := s5t#40s, Q => #_w1);
   "Tag_75" := #_w1;
END_REGION

REGION Network 15: запрет движения второй горки прокладок М314
   RUNG wire#powerrail
      Contact( "B17.2" )
      S_OFFDT(T_NO := "Tag_11", TV := s5t#2s, R :=, BI =>, RET_VAL =>)
      Coil( "Tag_70" )
   END_RUNG
   // the same network as SCL:
   #_s5time1 := S_OFFDT(T_NO := "Tag_11", S := "B17.2", TV := s5t#2s, Q => #_w1);
   "Tag_70" := #_w1;
END_REGION

REGION Network 16: Авто запуск второй горки прокладок М 314
   RUNG wire#powerrail
      Contact( "ALG".Auto_Gasket )
      I_Contact( "ALG".Alarm_Gasket )
      Contact( "Tag_75" )
      I_Contact( "Tag_70" )
      Coil( "IM".M_314_Second_slide.OnCom )
   END_RUNG
   // the same network as SCL:
   "IM".M_314_Second_slide.OnCom := "ALG".Auto_Gasket AND NOT "ALG".Alarm_Gasket AND "Tag_75" AND NOT "Tag_70";
END_REGION

REGION Network 17: Авто вперед третей горки прокладок M 315
   RUNG wire#powerrail
      Contact( "ALG".Auto_Gasket )
      I_Contact( "ALG".Alarm_Gasket )
      I_Contact( "Tag_112" )
      Contact( "Tag_57" )
      Coil( "IM".M_315_Third_slide.OnCom )
   END_RUNG
   // the same network as SCL:
   "IM".M_315_Third_slide.OnCom := "ALG".Auto_Gasket AND NOT "ALG".Alarm_Gasket AND NOT "Tag_112" AND "Tag_57";
END_REGION

REGION Network 18: Тригер на разрешение движения третей горки прокладок М315
   RUNG wire#powerrail
      Contact( "B17.2" )
      I_Contact( "Tag_124" )
      S_SR(operand := #Trig315, r1 := wire#w1)
      Coil( "Tag_57" )
   END_RUNG
   RUNG wire#powerrail
      Contact( "Tag_48" )
   END_RUNG wire#w1
   // the same network as SCL:
   IF "B17.2" AND NOT "Tag_124" THEN
       #Trig315 := TRUE;   // SR flip-flop
   END_IF;
   IF "Tag_48" THEN #Trig315 := FALSE; END_IF;
   "Tag_57" := #Trig315;
END_REGION

REGION Network 19: Авто вперед транспортер под крюками прокладок M234
   RUNG wire#powerrail
      Contact( "ALG".Auto_Sorting )
      I_Contact( "Tag_112" )
      Coil( "IM".M_234_Carousel_loader.OnCom )
   END_RUNG
   // the same network as SCL:
   "IM".M_234_Carousel_loader.OnCom := "ALG".Auto_Sorting AND NOT "Tag_112";
END_REGION

REGION Network 20: Задержка на датчик максимального слоя прокладки 234.2
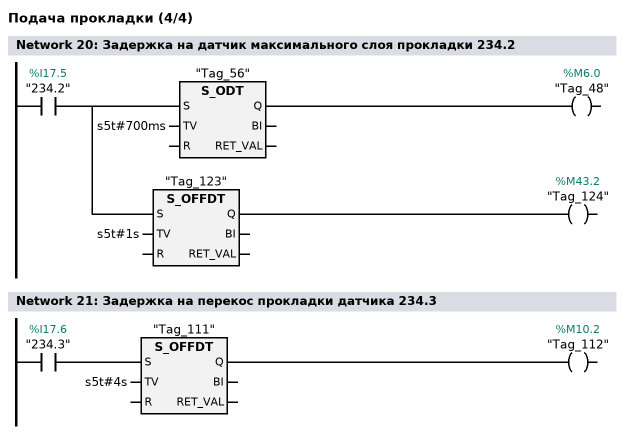
   RUNG wire#powerrail
      Contact( "234.2" )
      wire#w1
      S_ODT(T_NO := "Tag_56", TV := s5t#700ms, R :=, BI =>, RET_VAL =>)
      Coil( "Tag_48" )
   END_RUNG
   RUNG wire#w1
      S_OFFDT(T_NO := "Tag_123", TV := s5t#1s, R :=, BI =>, RET_VAL =>)
      Coil( "Tag_124" )
   END_RUNG
   // the same network as SCL:
   #_w2 := "234.2";
   #_s5time1 := S_ODT(T_NO := "Tag_56", S := "234.2", TV := s5t#700ms, Q => #_w1);
   "Tag_48" := #_w1;
   #_s5time2 := S_OFFDT(T_NO := "Tag_123", S := #_w2, TV := s5t#1s, Q => #_w3);
   "Tag_124" := #_w3;
END_REGION

REGION Network 21: Задержка на перекос прокладки датчика 234.3
   RUNG wire#powerrail
      Contact( "234.3" )
      S_OFFDT(T_NO := "Tag_111", TV := s5t#4s, R :=, BI =>, RET_VAL =>)
      Coil( "Tag_112" )
   END_RUNG
   // the same network as SCL:
   #_s5time1 := S_OFFDT(T_NO := "Tag_111", S := "234.3", TV := s5t#4s, Q => #_w1);
   "Tag_112" := #_w1;
END_REGION
END_FUNCTION_BLOCK

FUNCTION_BLOCK "FB_Rollout_Zone"
{ S7_Optimized_Access := 'FALSE' }
VERSION : 0.1
   VAR_INPUT 
      lift_returning : Bool;
      packet_ready : Bool;
      m_322_sensor : Bool;
      m_324_sensor : Bool;
      m_324_sync : Bool;
      lift_down_sensor : Bool;
      lift_up_sensor : Bool;
   END_VAR

   VAR_OUTPUT 
      packet_released : Bool;
   END_VAR

   VAR_IN_OUT 
      rolling_packet { ExternalAccessible := 'False'; ExternalVisible := 'False'; ExternalWritable := 'False'} : Bool;
   END_VAR

   VAR 
      busyM321 : Bool;
      busyM322 : Bool;
      busyM322_old : Bool;
      busyM324 : Bool;
      m_324_ready : Bool;
      m_324_move_trig : Bool;
      m_324_sens_old : Bool;
      m_324_sync_old : Bool;
      safe_rollout_timer {InstructionName := 'TON'; LibVersion := '1.0'; S7_SetPoint := 'False'} : TON;
      delay_start_m_324 {InstructionName := 'TON'; LibVersion := '1.0'} : TON;
      busy321_timer {InstructionName := 'TON'; LibVersion := '1.0'} : TON;
      busy322_timer {InstructionName := 'TOF'; LibVersion := '1.0'} : TOF;
      busy324_timer {InstructionName := 'TOF'; LibVersion := '1.0'} : TOF;
   END_VAR

   VAR_TEMP 
      packet_is_picked : Bool;
      rollout_ready : Bool;
   END_VAR

   VAR CONSTANT 
      ROLL_TIMEOUT : Time := T#4s;
      DELAY_START_324 : Time := T#3500ms;
   END_VAR


BEGIN
	REGION Ready and alarms ROLLOUT ZONE
	    "ALG".Ready_Rout := "NaprUpr" AND "K1-112 2L1" AND "K1-113/3 5L1";
	    
	    "ALG".Alarm_Rout :=
	    // Рольганг на лифте
	    "IM_Rout".M_321_Rollgang_Lift_PFM.Fault OR
	    "IM_Rout".M_321_Rollgang_Lift_PFM.Alarm OR
	    // Второй конвейер
	    "IM_Rout".M_322_Conveyor_2.Fault OR
	    "IM_Rout".M_322_Conveyor_2.Alarm OR
	    // Последний конвейер
	    "IM_Rout".M_324_Rout_Conveyor.Fault OR
	    "IM_Rout".M_324_Rout_Conveyor.Alarm OR
	    // Нет сигнала готовности
	    NOT "ALG".Ready_Rout;
	    
	    
	END_REGION
	
	REGION SIGNALS
	    #busy321_timer(IN := #lift_down_sensor,
	                   PT := T#2s,
	                   Q => #busyM321);
	    
	    #busy322_timer(IN := #m_322_sensor,
	                   PT := T#2s,
	                   Q => #busyM322);
	    
	    
	    #busy324_timer(IN := #m_324_sensor,
	                   PT := T#15s,
	                   Q => #busyM324);
	    
	    #packet_is_picked := #busyM322 AND NOT #busyM322_old;
	    
	    #busyM322_old := #busyM322;
	    
	END_REGION
	
	REGION Connection with MAIN SORTER
	    
	    #safe_rollout_timer(IN := #rolling_packet,
	                        PT := #ROLL_TIMEOUT);
	    
	    
	    IF (#rolling_packet AND #safe_rollout_timer.Q AND #packet_is_picked) THEN
	        #rolling_packet := FALSE;
	        
	        #packet_released := TRUE;
	    END_IF;
	    
	    IF (#packet_released AND ((#lift_returning AND NOT #lift_down_sensor) OR #lift_up_sensor)) THEN
	        #packet_released := FALSE;
	        
	    END_IF;
	    
	    // NEW feature
	    IF (#packet_ready AND NOT #lift_down_sensor) THEN
	        #rolling_packet := FALSE;
	    END_IF;
	   
	   
	END_REGION
	
	
	REGION helper values
	    
	    // нормальные условия для работы
	    #rollout_ready := NOT "ALG".Alarm_Rout AND "ALG".Auto_Sorting;
	    
	    // верное положение транспортера
	    #m_324_ready := (#m_324_ready OR
	    (
	    (#m_324_sync AND NOT #m_324_sync_old)
	    )
	    ) AND NOT (
	    (NOT #m_324_sensor AND #m_324_sens_old)
	    );
	    
	    #m_324_sync_old := #m_324_sync;
	    #m_324_sens_old := #m_324_sensor;
	    
	    
	END_REGION
	
	
	REGION Automode M321
	    
	    "IM_Rout".M_321_Rollgang_Lift_PFM.OnCom :=
	    
	    #rollout_ready AND
	        #rolling_packet AND
	        #busyM321 AND
	        NOT #busyM322;
	    
	END_REGION
	
	
	
	REGION Automode 322
	    
	    "IM_Rout".M_322_Conveyor_2.OnCom :=
	    
	    #rollout_ready AND
	    (
	    (
	    #busyM322 AND // есть пакет на 322
	    #m_324_ready AND // 324 в верном положении
	    NOT #busyM324 // свободен 324
	    )
	    OR
	    (
	    NOT #busyM322 AND // свободен 322
	    #busyM321 AND // есть пакет на 321
	    #rolling_packet // лифт заблокирован и дает разрешение на выкатку
	    )
	    );
	    
	END_REGION
	
	
	REGION Automode 324
	    
	    // захват движения M324
	    // 
	    #m_324_move_trig := (#m_324_move_trig OR
	    (
	    #busyM322 AND
	    #m_324_ready AND
	    NOT #busyM324
	    )
	    ) AND NOT (
	    #busyM324
	    );
	    
	    
	    // задержка на старт по условию
	    #delay_start_m_324(IN := #m_324_move_trig,
	                       PT := #DELAY_START_324);
	    
	    
	    "IM_Rout".M_324_Rout_Conveyor.OnCom :=
	    
	    #rollout_ready AND
	    NOT #busyM324 AND
	    (
	    NOT #m_324_ready OR #delay_start_m_324.Q
	    );
	    
	    
	    
	    // ПЧ 324
	    // DEPRECATED
	    IF ("IM_Rout".M_324_Rout_Conveyor.onOutBWD OR "IM_Rout".M_324_Rout_Conveyor.onOutFWD) THEN
	        "IM_Rout".M_324_Rout_Conveyor.setSpeedAU := 8.0;
	    ELSE
	        "IM_Rout".M_324_Rout_Conveyor.setSpeedAU := 0.0;
	    END_IF;
	    
	END_REGION
	
END_FUNCTION_BLOCK

FUNCTION_BLOCK "FB_Gasket_Carousel"
{ S7_Optimized_Access := 'FALSE' }
VERSION : 0.1
   VAR_INPUT 
      make_layer : Bool;
      may_release : Bool;
      full_reset : Bool;
      pause : Bool;
      try_unpause : Bool;
      gasket_sensor : Bool;
      hook_sensor : Bool;
      last_hook_sensor : Bool;
      no_ramp_flag : Bool;
      enable_double_schema : Bool;
      layer_num : Int;
      "2_schema_height" : Int;
      GASKET_PLACES_MAX : Int;
      HOOK_ENCODER_BARRIER : Int := 40;
      GUARANTEED_HOOK_OFFSET : Int := 250;
      OFFSET_DOWN_DEVICE : Int;
      OFFSET_LAST_HOOK : Int;
      OFFSET_LAYER_READY : Int;
      OFFSET_REVERS : Int;
      enc_pos : DInt;
      "1_schema_server" : DInt;
      "2_schema_server" : DInt;
      default_speed : Real;
      offset_speed : Real;
      default_reverse_speed : Real;
   END_VAR

   VAR_OUTPUT 
      Carousel_FWD : Bool;
      Carousel_BWD : Bool;
      Ski_UP : Bool;
      Ski_DOWN : Bool;
      m_busy : Bool;
      m_acquire : Bool;
      m_released : Bool;
      ALM_NoGasketToUP : Bool;
      ALM_SensHook : Bool;
      ALM_SensLastHook : Bool;
      s_man_cntl : Bool;
      s_paused : Bool;
      s_reset_encoder : Bool;
      Carousel_Speed : Real;
   END_VAR

   VAR 
      pos_defined : Bool;
      gasket_ready : Bool;
      _State : Int;
      s_max_hooks : Int;
      schema : DInt;
      SX { ExternalAccessible := 'False'; ExternalVisible := 'False'; ExternalWritable := 'False'} AT schema : Array[0..31] of Bool;
      enc_shot : DInt;
      hook_hold_timer {InstructionName := 'TOF'; LibVersion := '1.0'; S7_SetPoint := 'False'} : TOF;
      last_hook_hold_timer {InstructionName := 'TOF'; LibVersion := '1.0'} : TOF;
      gasket_filter {InstructionName := 'TON'; LibVersion := '1.0'} : TON;
      Counters : Struct   // inner counters
         hooks : Int;
      END_STRUCT;
      Memento : Struct   // memento pattern
         fwd : Bool;
         bwd : Bool;
         up : Bool;
         down : Bool;
         state : Int;
         speed : Real;
      END_STRUCT;
      SIG_old : Struct
         hook : Bool;
         last_hook : Bool;
      END_STRUCT;
   END_VAR

   VAR_TEMP 
      valid_hook : Bool;
      corrected_state : Bool;
      index : Int;
      hook_period_pos : DInt;
      SIG : Struct
         new_hook : Bool;
         last_hook : Bool;
      END_STRUCT;
   END_VAR

   VAR CONSTANT 
      STATE_WAITING : Int := 0;
      STATE_CYCLE : Int := 3;
      STATE_NO_MORE_GASKET : Int := 4;
      STATE_POSITIONING : Int := 5;
      STATE_FULL : Int := 7;
      STATE_RELEASE : Int := 9;
      STATE_MAN_CORRECT : Int := 11;
      STATE_AUTO_CORRECT : Int := 13;
      STATE_PAUSE : Int := 100;
   END_VAR


BEGIN
	REGION Timers Delays
	    #hook_hold_timer(IN := #hook_sensor,
	                     PT := T#600ms);
	    
	    #gasket_filter(IN := #gasket_sensor,
	                   PT := T#2s);
	    
	END_REGION
	
	REGION SIGNALS
	    // hot signals
	    #SIG.new_hook := #hook_hold_timer.Q AND NOT #SIG_old.hook;
	    #SIG.last_hook := #last_hook_sensor AND NOT #SIG_old.last_hook;
	    
	    
	    // old signals
	    #SIG_old.hook := #hook_hold_timer.Q;
	    #SIG_old.last_hook := #last_hook_sensor;
	END_REGION
	
	
	REGION Helpers
	    
	    #gasket_ready := (#gasket_ready OR
	    (
	    #gasket_filter.ET >= T#100ms
	    )) AND NOT (
	    #Ski_UP
	    );
	    
	    #hook_period_pos := #enc_pos - #enc_shot;
	    
	END_REGION
	
	
	REGION non-case restart and pause
	    IF (#pause AND NOT #s_paused) THEN
	        #Memento.state := #_State;
	        
	        #s_paused := TRUE;
	        
	        #_State := #STATE_PAUSE;
	    END_IF;
	    
	    IF (#full_reset) THEN
	        #_State := #STATE_WAITING;
	    END_IF;
	    
	END_REGION
	
	
	REGION Reset output flags
	    #s_reset_encoder := FALSE;
	END_REGION
	
	StartAutomat:
	CASE #_State OF
	    #STATE_WAITING:
	        // Logic
	        #Carousel_FWD := FALSE;
	        #Carousel_BWD := FALSE;
	        #Ski_UP := FALSE;
	        #Ski_DOWN := TRUE;
	        
	        #m_busy := FALSE; // флаг занятости карусели
	        #m_acquire := FALSE; // флаг возможности захвата прокладок
	        
	        #s_paused := FALSE;
	        #s_man_cntl := FALSE;
	        
	        // select schema
	        IF (#layer_num < #"2_schema_height" AND #enable_double_schema) THEN
	            #schema := #"2_schema_server";
	        ELSE
	            #schema := #"1_schema_server";
	        END_IF;
	        
	        // reset alarms
	        // 
	        #ALM_SensHook := false;
	        #ALM_SensLastHook := FALSE;
	        #ALM_NoGasketToUP := FALSE;
	        
	        #pos_defined := FALSE;
	        
	        #Counters.hooks := 0;
	        #Carousel_Speed := 0.0;
	        
	        // transitions
	        // 
	        IF (#make_layer AND #no_ramp_flag) THEN
	            #_State := #STATE_CYCLE;
	            #m_busy := TRUE;
	            #m_released := FALSE; // можно ли опускать каретку
	            
	            #s_max_hooks := "getMaxBit"(MAX:=#GASKET_PLACES_MAX, number:=#schema);
	            
	            // сбрасываем счетчик энкодера
	            // 
	            #s_reset_encoder := TRUE;
	            
	        END_IF;
	    
	    #STATE_CYCLE:
	        // Logic
	        #Carousel_FWD := TRUE;
	        #Carousel_BWD := FALSE;
	        
	        #Carousel_Speed := #default_speed;
	        
	        REGION helpers
	            // Необходимость привода индекса из-за обратного порядка битов в байте числа Sxema
	            // сначала по нужному нам индексу в числе понимаем, какой нужен байт: (11 + hookcounter) div 8
	            // сдвиг на 11 потому что старшие 11 битов не нужны (всего 21 ложемент)
	            // далее учтем обратный порядок битов в этом байте
	            // нужный бит будет иметь позицию 7 - (11 + hookcounter) mod 8
	            // теперь добавим данный номер бита к номеру байта и получим нужную позицию в числе
	            // после упрощений получим результат:
	            #index := 18 + #Counters.hooks - 2 * ((11 + #Counters.hooks) MOD 8);
	            
	            #valid_hook := (ABS_DINT(#hook_period_pos) >= #HOOK_ENCODER_BARRIER) OR (NOT #pos_defined);
	            
	        END_REGION
	        
	        //throw hook error
	        #ALM_SensHook := #pos_defined AND (#hook_period_pos >= #GUARANTEED_HOOK_OFFSET);
	        
	        IF (#ALM_SensHook) THEN
	            // заполняем структуру состояния
	            // 
	            #Memento.state := #_State;
	            
	            #_State := #STATE_MAN_CORRECT;
	            GOTO EndMAchine;
	        END_IF;
	        
	        
	        // TODO: check conditions!!!!!
	        // 
	        // если лыжи надо опустить (они подняты) и проехали нужное расстояние
	        IF (#Ski_UP) THEN
	            IF (#hook_period_pos >= #OFFSET_DOWN_DEVICE) THEN
	                // опускаем лыжи
	                #Ski_UP := FALSE;
	                #Ski_DOWN := TRUE;
	            END_IF;
	        ELSIF (#SIG.new_hook AND #valid_hook) THEN
	            IF (#Counters.hooks < #GASKET_PLACES_MAX) THEN
	                
	                #ALM_NoGasketToUP := #SX[#index] AND NOT #gasket_ready;
	                
	                #Counters.hooks := #Counters.hooks + 1;
	                
	                #pos_defined := TRUE;
	                #enc_shot := #enc_pos;
	                
	                #Ski_UP := #SX[#index] AND #gasket_ready;
	                #Ski_DOWN := FALSE;
	                
	            END_IF;
	           
	           
	        END_IF;
	        
	        // TEST!!! Ускорение
	        IF (#Counters.hooks > #s_max_hooks AND NOT #Ski_UP) THEN
	            #Carousel_Speed := #offset_speed;
	        END_IF;
	        
	        // transitions
	        IF (#ALM_NoGasketToUP) THEN
	            #Memento.state := #_State;
	            
	            #_State := #STATE_AUTO_CORRECT;
	            GOTO EndMAchine;
	            
	            // Если все ложементы прошли и опустили лыжи
	        ELSIF (#Counters.hooks = #GASKET_PLACES_MAX AND NOT #Ski_UP) THEN
	            #_State := #STATE_POSITIONING;
	            
	        END_IF;
	        
	    #STATE_NO_MORE_GASKET:
	        ;
	        
	    #STATE_POSITIONING:
	        // logic
	        #Carousel_FWD := TRUE;
	        #Carousel_BWD := FALSE;
	        
	        #Carousel_Speed := 6.5;
	        
	        #Ski_UP := FALSE;
	        #Ski_DOWN := TRUE;
	        
	        // throw error
	        #ALM_SensLastHook := (#hook_period_pos >= #OFFSET_LAYER_READY);
	        
	        // transitions
	        IF (#ALM_SensLastHook) THEN
	            // заполняем структуру состояния
	            #Memento.state := #_State;
	            
	            #_State := #STATE_MAN_CORRECT;
	            GOTO EndMAchine;
	        END_IF;
	        
	        (*
	        // helper
	        // 
	        //#valid_hook := ABS_DINT(#hook_period_pos) >= #HOOK_ENCODER_BARRIER;
	        
	        // прошел сенсор
	        IF () THEN
	            #Counters.hooks := #Counters.hooks + 1;
	            #Carousel_Speed := 0.7 * #Carousel_Speed;
	        END_IF;
	        
	        IF (#Counters.hooks = #index) THEN
	            #_State := #STATE_FULL;
	            #Carousel_FWD := False;
	        END_IF; *)
	        
	        IF (#SIG.last_hook AND #hook_period_pos >= #OFFSET_LAST_HOOK) THEN
	            
	                #_State := #STATE_FULL;
	                #Carousel_FWD := FALSE;
	
	        END_IF;
	        
	        
	        
	    #STATE_FULL:
	        
	        #Carousel_BWD := FALSE;
	        #Carousel_FWD := False;
	        #Carousel_Speed := 0.0;
	        
	        #m_acquire := TRUE; // забирайте прокладки ради Бога флаг захвата выставлен
	        #m_released := FALSE;
	        
	        // если каретка приехала с закрытыми ложементами можно отъезжать
	        IF ( #may_release ) THEN
	            #_State := #STATE_RELEASE;
	            // снапшот
	            // 
	            #Counters.hooks := 0;
	            #enc_shot := #enc_pos;
	            #m_acquire := FALSE;
	        END_IF;
	        
	        
	    #STATE_RELEASE:
	        #m_acquire := FALSE;
	        
	        #Carousel_BWD := TRUE;
	        #Carousel_FWD := FALSE;
	        
	        #Carousel_Speed := #default_reverse_speed;
	        
	        IF (-#hook_period_pos >= #OFFSET_REVERS AND NOT #last_hook_sensor) THEN
	            #Carousel_BWD := FALSE;
	            #m_released := TRUE;
	            #_State := #STATE_WAITING;
	            GOTO EndMAchine;
	        END_IF;
	        
	        
	    #STATE_MAN_CORRECT:
	        // даем ручное управление оператору
	        #s_man_cntl := TRUE;
	        #s_paused := TRUE;
	        
	        #Carousel_FWD := FALSE;
	        #Carousel_BWD := FALSE;
	        #Carousel_Speed := 0.0;
	        
	        // оператор выровнял крюк и датчик
	        #corrected_state :=
	        (#ALM_SensHook AND #hook_sensor)
	        OR
	        (#ALM_SensLastHook AND #last_hook_sensor);
	        
	        IF (#corrected_state AND #try_unpause) THEN
	            
	            // вернем состояние
	            // 
	            #_State := #Memento.state;
	            #s_man_cntl := false;
	            #s_paused := FALSE;
	            
	            // убиваем ошибки
	            // 
	            #ALM_SensHook := FALSE;
	            #ALM_SensLastHook := FALSE;
	            
	            // создаем фронт для датчика
	            // 
	            #SIG_old.hook := FALSE;
	            #SIG_old.last_hook := False;
	            
	        END_IF;
	        
	        
	    #STATE_AUTO_CORRECT:
	        
	        #s_paused := TRUE;
	        
	        #Carousel_FWD := FALSE;
	        #Carousel_BWD := FALSE;
	        #Carousel_Speed := 0.0;
	        
	        #Ski_DOWN := TRUE;
	        #Ski_UP := FALSE;
	        
	        // если при ошибке отсутсвия рейки рейка появилась то поднимем девайс и снимем паузу
	        IF (#ALM_NoGasketToUP AND #gasket_ready) THEN
	            #Ski_UP := TRUE;
	            #Ski_DOWN := FALSE;
	            
	            #ALM_NoGasketToUP := FALSE;
	            
	            #s_paused := FALSE;
	            
	            #_State := #Memento.state;
	        END_IF;
	        
	    #STATE_PAUSE:
	        // ставим карусель на паузу
	        #s_paused := TRUE;
	        
	        #Carousel_FWD := FALSE;
	        #Carousel_BWD := FALSE;
	        #Carousel_Speed := 0.0;
	        
	        IF (NOT #pause) THEN
	            #_State := #Memento.state;
	            
	            #s_paused := False;
	        END_IF;
	        
	END_CASE;
	
	EndMAchine:
	RETURN;
END_FUNCTION_BLOCK

FUNCTION "getMaxBit" : Int
{ S7_Optimized_Access := 'FALSE' }
VERSION : 0.1
   VAR_INPUT 
      MAX : Int;
      number : DInt;
   END_VAR

   VAR_TEMP 
      index : Int;
      i : Int;
      num : DInt;
      SX AT num : Array[0..31] of Bool;
   END_VAR


BEGIN
	// naive
	// 
	#num := #number;
	
	FOR #i := #MAX - 1 TO 0 BY -1 DO
	    // Необходимость привода индекса из-за обратного порядка битов в байте числа Sxema
	    // сначала по нужному нам индексу в числе понимаем, какой нужен байт: (11 + hookcounter) div 8
	    // сдвиг на 11 потому что старшие 11 битов не нужны (всего 21 ложемент)
	    // далее учтем обратный порядок битов в этом байте
	    // нужный бит будет иметь позицию 7 - (11 + hookcounter) mod 8
	    // теперь добавим данный номер бита к номеру байта и получим нужную позицию в числе
	    // после упрощений получим результат:
	    #index := 18 + #i - 2 * ((11 + #i) MOD 8);
	    IF (#SX[#index]) THEN
	        EXIT;
	    END_IF;
	END_FOR;
	
	
	#getMaxBit := #i;
	
END_FUNCTION

FUNCTION_BLOCK "Сортировка"   // FB9, LAD
VERSION : 0.1
// Логика работы ПФМ
// stored: AutoNumber true, IsIECCheckEnabled false, UDAEnableTagReadback false
   VAR_INPUT
      packet_released : Bool;
   END_VAR
   VAR DB_SPECIFIC
      "TrigE76.4" : Bool;
      Trig_Dovod : Bool;
      LiftPushingPacket : Bool;
      TrigAutoPFM : Bool;
      Trig_Vill : Bool;
      Trig_Vill2 : Bool;
      LiftDownTrig : Bool;
      HaveSxema : Bool;
      NewPacket : Bool;
      LiftDown_old : Bool;
      LiftPushing_old : Bool;
      ForksForcingFinish : Bool;
      LiftForcingFinish : Bool;
      CommonForcingPacket : Bool;
      ElevatorLowering : Bool;
      NoGasketMode : Bool;   // режим без прокладки
      RampIsOn : Bool;
      RampIsOff : Bool;
      power_Vill : Bool := true;
      MakedLayer : Bool;
      AlarmLowerElevator : Bool;
      AlarmNotReadedPack : Bool;
      lift_return_trig : Bool;
      ramp_sync_old : Bool;
      BoardInLayerCounter : Int;
      LayersCounter : Int;
   END_VAR
   VAR
      Vibrator_KeyFazer { S7_SetPoint := 'True'} : "Vibrator";
      Run323_timer { S7_SetPoint := 'True'} : TP;
      LayerCounter { S7_SetPoint := 'True'} : "Adder";
   END_VAR
   VAR_TEMP
      Sert : Word;
   END_VAR
   VAR_TEMP   // added for the SCL form of the ladder/FBD networks
      _w1 : Bool;
      _w2 : Bool;
      _s5time1 : S5Time;
      _w3 : Bool;
      _w4 : Bool;
      _w5 : Bool;
      _s5time2 : S5Time;
   END_VAR
BEGIN

REGION Network 1: 221 группа на 14 моторов общий сигнал готовности
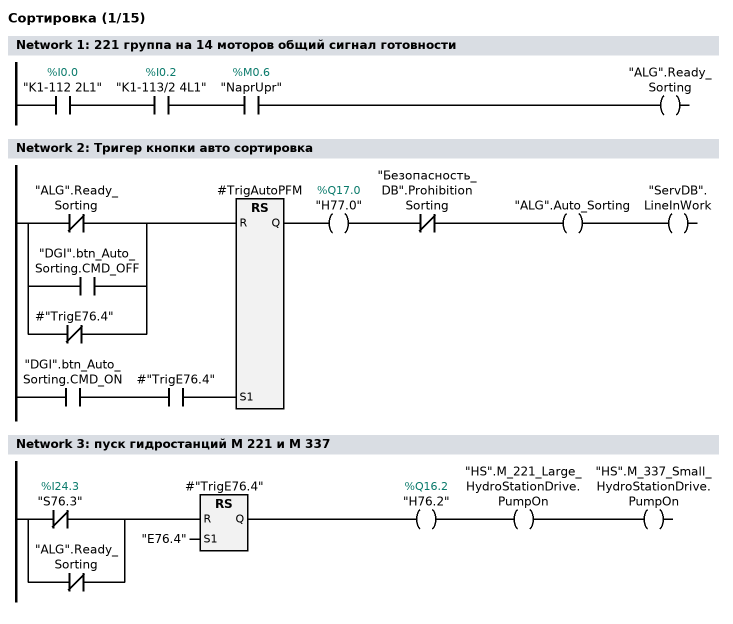
   RUNG wire#powerrail
      Contact( "K1-112 2L1" )
      Contact( "K1-113/2 4L1" )
      Contact( "NaprUpr" )
      Coil( "ALG".Ready_Sorting )
   END_RUNG
   // the same network as SCL:
   "ALG".Ready_Sorting := "K1-112 2L1" AND "K1-113/2 4L1" AND "NaprUpr";
END_REGION

REGION Network 2: Тригер кнопки авто сортировка
   RUNG wire#powerrail
      I_Contact( "ALG".Ready_Sorting )
      wire#w1
      S_RS(operand := #TrigAutoPFM, s1 := wire#w2)
      Coil( "H77.0" )
      I_Contact( "Безопасность_DB".ProhibitionSorting )
      Coil( "ALG".Auto_Sorting )
      Coil( "ServDB".LineInWork )
   END_RUNG
   RUNG wire#powerrail
      Contact( "DGI".btn_Auto_Sorting.CMD_OFF )
   END_RUNG wire#w1
   RUNG wire#powerrail
      I_Contact( #"TrigE76.4" )
   END_RUNG wire#w1
   RUNG wire#powerrail
      Contact( "DGI".btn_Auto_Sorting.CMD_ON )
      Contact( #"TrigE76.4" )
   END_RUNG wire#w2
   // the same network as SCL:
   IF NOT "ALG".Ready_Sorting OR "DGI".btn_Auto_Sorting.CMD_OFF OR NOT #"TrigE76.4" THEN
       #TrigAutoPFM := FALSE;   // RS flip-flop
   END_IF;
   IF "DGI".btn_Auto_Sorting.CMD_ON AND #"TrigE76.4" THEN #TrigAutoPFM := TRUE; END_IF;
   "H77.0" := #TrigAutoPFM;
   "ALG".Auto_Sorting := #TrigAutoPFM AND NOT "Безопасность_DB".ProhibitionSorting;
   "ServDB".LineInWork := "ALG".Auto_Sorting;
END_REGION

REGION Network 3: пуск гидростанций М 221 и M 337
   RUNG wire#powerrail
      I_Contact( "S76.3" )
      wire#w1
      S_RS(operand := #"TrigE76.4", s1 := "E76.4")
      Coil( "H76.2" )
      Coil( "HS".M_221_Large_HydroStationDrive.PumpOn )
      Coil( "HS".M_337_Small_HydroStationDrive.PumpOn )
   END_RUNG
   RUNG wire#powerrail
      I_Contact( "ALG".Ready_Sorting )
   END_RUNG wire#w1
   // the same network as SCL:
   IF NOT "S76.3" OR NOT "ALG".Ready_Sorting THEN
       #"TrigE76.4" := FALSE;   // RS flip-flop
   END_IF;
   IF "E76.4" THEN #"TrigE76.4" := TRUE; END_IF;
   "H76.2" := #"TrigE76.4";
   "HS".M_221_Large_HydroStationDrive.PumpOn := #"TrigE76.4";
   "HS".M_337_Small_HydroStationDrive.PumpOn := #"TrigE76.4";
END_REGION

